C01761=-95.203,-21.462,17.374,-169.9520,-5.2148,-3137.2959
C01762=-94.842,-19.790,17.237,-164.8285,-6.4355,-3138.2136
C01763=-94.656,-17.748,17.095,-159.3411,-5.0626,-3139.3803
C01764=-94.777,-14.774,16.986,-155.9417,-1.9916,-3141.1399
C01765=-95.219,-10.339,16.941,-154.9335,-0.3011,-3143.8030
C01766=-95.617,-5.406,16.939,-154.8750,0.0274,-3146.7641
C01767=-95.772,0.000,16.941,-154.8879,-0.0000,-3150.0000
C01768=-95.617,5.406,16.939,-154.8750,-0.0274,-3153.2359
C01769=-95.219,10.339,16.941,-154.9335,0.3011,-3156.1970
C01770=-94.777,14.774,16.986,-155.9409,1.9854,-3158.8601
C01771=-94.656,17.748,17.095,-159.3411,5.0626,-3160.6197
C01772=-94.842,19.790,17.237,-164.8285,6.4355,-3161.7864
C01773=-95.203,21.462,17.374,-169.9520,5.2148,-3162.7041
C01774=-95.565,23.155,17.473,-173.2181,2.8849,-3163.6200
C01775=-95.708,25.257,17.521,-175.7539,1.0630,-3164.7831
C01776=-95.481,28.035,17.545,-178.1294,0.2806,-3166.3632
C01777=-94.884,31.135,17.565,-179.6411,0.0273,-3168.1666
C01778=-93.972,34.135,17.585,-179.9202,-0.0015,-3169.9634
C01779=-92.934,36.917,17.598,-179.9926,-0.0032,-3171.6649
C01780=-91.818,39.610,17.598,-179.9925,-0.0030,-3173.3352
C01781=-90.585,42.311,17.585,-179.9180,0.0004,-3175.0366
C01782=-89.109,45.077,17.565,-179.6386,-0.0291,-3176.8332
C01783=-87.339,47.692,17.545,-178.1307,-0.2787,-3178.6370
C01784=-85.535,49.816,17.521,-175.7503,-1.0646,-3180.2167
C01785=-83.948,51.202,17.473,-173.2162,-2.8847,-3181.3801
C01786=-82.495,52.143,17.374,-169.9475,-5.2185,-3182.2959
C01787=-81.058,53.070,17.237,-164.8269,-6.4371,-3183.2134
C01788=-79.482,54.382,17.095,-159.3399,-5.0676,-3184.3801
C01789=-77.464,56.571,16.986,-155.9409,-1.9875,-3186.1402
C01790=-74.640,60.019,16.941,-154.9325,-0.3004,-3188.8032
C01791=-71.434,63.789,16.939,-154.8745,0.0271,-3191.7642
C01792=-67.721,67.721,16.941,-154.8876,0.0000,-3195.0000
C01793=-63.789,71.434,16.939,-154.8745,-0.0271,-3198.2358
C01794=-60.019,74.640,16.941,-154.9325,0.3004,-3201.1968
C01795=-56.571,77.464,16.986,-155.9409,1.9875,-3203.8598
C01796=-54.382,79.482,17.095,-159.3399,5.0676,-3205.6199
C01797=-53.070,81.058,17.237,-164.8269,6.4371,-3206.7866
C01798=-52.143,82.495,17.374,-169.9475,5.2185,-3207.7041
C01799=-51.202,83.948,17.473,-173.2162,2.8847,-3208.6199
C01800=-49.816,85.535,17.521,-175.7503,1.0646,-3209.7833
C01801=-47.692,87.339,17.545,-178.1307,0.2787,-3211.3630
C01802=-45.077,89.109,17.565,-179.6386,0.0291,-3213.1668
C01803=-42.311,90.585,17.585,-179.9180,-0.0004,-3214.9634
C01804=-39.610,91.818,17.598,-179.9925,0.0030,-3216.6648
C01805=-36.917,92.934,17.598,-179.9926,0.0032,-3218.3351
C01806=-34.135,93.972,17.585,-179.9202,0.0015,-3220.0366
C01807=-31.135,94.884,17.565,-179.6411,-0.0273,-3221.8334
C01808=-28.035,95.481,17.545,-178.1294,-0.2806,-3223.6368
C01809=-25.257,95.708,17.521,-175.7539,-1.0630,-3225.2169
C01810=-23.155,95.565,17.473,-173.2181,-2.8849,-3226.3800
C01811=-21.462,95.203,17.374,-169.9520,-5.2148,-3227.2959
C01812=-19.790,94.842,17.237,-164.8285,-6.4355,-3228.2136
C01813=-17.748,94.656,17.095,-159.3411,-5.0626,-3229.3803
C01814=-14.774,94.777,16.986,-155.9409,-1.9854,-3231.1399
C01815=-10.339,95.219,16.941,-154.9335,-0.3011,-3233.8030
C01816=-5.406,95.617,16.939,-154.8750,0.0274,-3236.7641
C01817=0.000,95.772,16.941,-154.8879,-0.0000,-3240.0000
C01818=0.000,94.804,18.916,-152.9225,-0.0000,-3240.0000
C01819=5.317,94.652,18.914,-152.9126,-0.0298,-3243.2152
C01820=10.190,94.262,18.917,-152.9815,0.4089,-3246.1699
C01821=14.592,93.857,18.976,-154.1276,2.6863,-3248.8371
C01822=17.528,93.824,19.120,-158.3516,6.7345,-3250.5819
C01823=19.540,94.146,19.309,-165.0906,8.0389,-3251.7253
C01824=21.192,94.676,19.493,-170.7538,6.1439,-3252.6169
C01825=22.867,95.222,19.627,-173.7811,3.3954,-3253.5035
C01826=24.945,95.538,19.692,-175.9706,1.2792,-3254.6333
C01827=27.741,95.446,19.726,-178.2555,0.3221,-3256.2063
C01828=30.903,94.927,19.753,-179.7244,0.0234,-3258.0324
C01829=33.988,94.020,19.780,-179.9222,0.0038,-3259.8748
C01830=36.867,92.953,19.798,-179.9926,-0.0032,-3261.6343
C01831=39.659,91.796,19.798,-179.9925,-0.0030,-3263.3660
C01832=42.449,90.515,19.780,-179.9232,-0.0019,-3265.1253
C01833=45.272,88.975,19.753,-179.7282,-0.0288,-3266.9678
C01834=47.874,87.106,19.726,-178.2537,-0.3220,-3268.7935
C01835=49.917,85.194,19.692,-175.9742,-1.2794,-3270.3670
C01836=51.163,83.502,19.627,-173.7835,-3.3967,-3271.4965
C01837=51.961,81.931,19.493,-170.7560,-6.1455,-3272.3830
C01838=52.755,80.388,19.309,-165.0938,-8.0387,-3273.2751
C01839=53.950,78.738,19.120,-158.3479,-6.7340,-3274.4183
C01840=56.048,76.685,18.976,-154.1288,-2.6854,-3276.1625
C01841=59.448,73.859,18.917,-152.9797,-0.4094,-3278.8301
C01842=63.169,70.689,18.914,-152.9124,0.0356,-3281.7846
C01843=67.036,67.036,18.916,-152.9207,0.0000,-3285.0000
C01844=70.689,63.169,18.914,-152.9124,-0.0356,-3288.2154
C01845=73.859,59.448,18.917,-152.9797,0.4094,-3291.1699
C01846=76.685,56.048,18.976,-154.1288,2.6854,-3293.8375
C01847=78.738,53.950,19.120,-158.3479,6.7340,-3295.5817
C01848=80.388,52.755,19.309,-165.0938,8.0387,-3296.7249
C01849=81.931,51.961,19.493,-170.7560,6.1455,-3297.6170
C01850=83.502,51.163,19.627,-173.7835,3.3967,-3298.5035
C01851=85.194,49.917,19.692,-175.9742,1.2794,-3299.6330
C01852=87.106,47.874,19.726,-178.2537,0.3220,-3301.2065
C01853=88.975,45.272,19.753,-179.7282,0.0288,-3303.0322
C01854=90.515,42.449,19.780,-179.9232,0.0019,-3304.8747
C01855=91.796,39.659,19.798,-179.9925,0.0030,-3306.6340
C01856=92.953,36.867,19.798,-179.9926,0.0032,-3308.3657
C01857=94.020,33.988,19.780,-179.9222,-0.0038,-3310.1252
C01858=94.927,30.903,19.753,-179.7244,-0.0234,-3311.9676
C01859=95.446,27.741,19.726,-178.2555,-0.3221,-3313.7937
C01860=95.538,24.945,19.692,-175.9706,-1.2792,-3315.3667
C01861=95.222,22.867,19.627,-173.7811,-3.3954,-3316.4965
C01862=94.676,21.192,19.493,-170.7538,-6.1439,-3317.3831
C01863=94.146,19.540,19.309,-165.0906,-8.0389,-3318.2747
C01864=93.824,17.528,19.120,-158.3516,-6.7345,-3319.4181
C01865=93.857,14.592,18.976,-154.1276,-2.6863,-3321.1629
C01866=94.262,10.190,18.917,-152.9815,-0.4089,-3323.8301
C01867=94.652,5.317,18.914,-152.9126,0.0298,-3326.7848
C01868=94.804,0.000,18.916,-152.9225,-0.0000,-3330.0000
C01869=94.652,-5.317,18.914,-152.9126,-0.0298,-3333.2152
C01870=94.262,-10.190,18.917,-152.9815,0.4089,-3336.1699
C01871=93.857,-14.592,18.976,-154.1276,2.6863,-3338.8371
C01872=93.824,-17.528,19.120,-158.3516,6.7345,-3340.5819
C01873=94.146,-19.540,19.309,-165.0906,8.0389,-3341.7253
C01874=94.676,-21.192,19.493,-170.7538,6.1439,-3342.6169
C01875=95.222,-22.867,19.627,-173.7811,3.3954,-3343.5035
C01876=95.538,-24.945,19.692,-175.9706,1.2792,-3344.6333
C01877=95.446,-27.741,19.726,-178.2555,0.3221,-3346.2063
C01878=94.927,-30.903,19.753,-179.7244,0.0234,-3348.0324
C01879=94.020,-33.988,19.780,-179.9222,0.0038,-3349.8748
C01880=92.953,-36.867,19.798,-179.9926,-0.0032,-3351.6343
C01881=91.796,-39.659,19.798,-179.9925,-0.0030,-3353.3660
C01882=90.515,-42.449,19.780,-179.9232,-0.0019,-3355.1253
C01883=88.975,-45.272,19.753,-179.7282,-0.0288,-3356.9678
C01884=87.106,-47.874,19.726,-178.2537,-0.3220,-3358.7935
C01885=85.194,-49.917,19.692,-175.9742,-1.2794,-3360.3670
C01886=83.502,-51.163,19.627,-173.7835,-3.3967,-3361.4965
C01887=81.931,-51.961,19.493,-170.7560,-6.1455,-3362.3830
C01888=80.388,-52.755,19.309,-165.0938,-8.0387,-3363.2751
C01889=78.738,-53.950,19.120,-158.3479,-6.7340,-3364.4183
C01890=76.685,-56.048,18.976,-154.1288,-2.6854,-3366.1625
C01891=73.859,-59.448,18.917,-152.9797,-0.4094,-3368.8301
C01892=70.689,-63.169,18.914,-152.9124,0.0356,-3371.7846
C01893=67.036,-67.036,18.916,-152.9207,-0.0000,-3375.0000
C01894=63.169,-70.689,18.914,-152.9124,-0.0356,-3378.2154
C01895=59.448,-73.859,18.917,-152.9797,0.4094,-3381.1699
C01896=56.048,-76.685,18.976,-154.1288,2.6854,-3383.8375
C01897=53.950,-78.738,19.120,-158.3479,6.7340,-3385.5817
C01898=52.755,-80.388,19.309,-165.0938,8.0387,-3386.7249
C01899=51.961,-81.931,19.493,-170.7560,6.1455,-3387.6170
C01900=51.163,-83.502,19.627,-173.7835,3.3967,-3388.5035
C01901=49.917,-85.194,19.692,-175.9742,1.2794,-3389.6330
C01902=47.874,-87.106,19.726,-178.2537,0.3220,-3391.2065
C01903=45.272,-88.975,19.753,-179.7282,0.0288,-3393.0322
C01904=42.449,-90.515,19.780,-179.9232,0.0019,-3394.8747
C01905=39.659,-91.796,19.798,-179.9925,0.0030,-3396.6340
C01906=36.867,-92.953,19.798,-179.9926,0.0032,-3398.3657
C01907=33.988,-94.020,19.780,-179.9222,-0.0038,-3400.1252
C01908=30.903,-94.927,19.753,-179.7244,-0.0234,-3401.9676
C01909=27.741,-95.446,19.726,-178.2555,-0.3221,-3403.7937
C01910=24.945,-95.538,19.692,-175.9706,-1.2792,-3405.3667
C01911=22.867,-95.222,19.627,-173.7811,-3.3954,-3406.4965
C01912=21.192,-94.676,19.493,-170.7538,-6.1439,-3407.3831
C01913=19.540,-94.146,19.309,-165.0906,-8.0389,-3408.2747
C01914=17.528,-93.824,19.120,-158.3516,-6.7345,-3409.4181
C01915=14.592,-93.857,18.976,-154.1276,-2.6863,-3411.1629
C01916=10.190,-94.262,18.917,-152.9815,-0.4089,-3413.8301
C01917=5.317,-94.652,18.914,-152.9126,0.0298,-3416.7848
C01918=0.000,-94.804,18.916,-152.9225,0.0000,-3420.0000
C01919=0.000,-94.804,18.916,-152.9225,0.0000,-3420.0000
C01920=-5.317,-94.652,18.914,-152.9126,-0.0298,-3423.2152
C01921=-10.190,-94.262,18.917,-152.9815,0.4089,-3426.1699
C01922=-14.592,-93.857,18.976,-154.1276,2.6863,-3428.8371
C01923=-17.528,-93.824,19.120,-158.3516,6.7345,-3430.5819
C01924=-19.540,-94.146,19.309,-165.0906,8.0389,-3431.7253
C01925=-21.192,-94.676,19.493,-170.7538,6.1439,-3432.6169
C01926=-22.867,-95.222,19.627,-173.7811,3.3954,-3433.5035
C01927=-24.945,-95.538,19.692,-175.9706,1.2792,-3434.6333
C01928=-27.741,-95.446,19.726,-178.2555,0.3221,-3436.2063
C01929=-30.903,-94.927,19.753,-179.7244,0.0234,-3438.0324
C01930=-33.988,-94.020,19.780,-179.9222,0.0038,-3439.8748
C01931=-36.867,-92.953,19.798,-179.9926,-0.0032,-3441.6343
C01932=-39.659,-91.796,19.798,-179.9925,-0.0030,-3443.3660
C01933=-42.449,-90.515,19.780,-179.9232,-0.0019,-3445.1253
C01934=-45.272,-88.975,19.753,-179.7282,-0.0288,-3446.9678
C01935=-47.874,-87.106,19.726,-178.2537,-0.3220,-3448.7935
C01936=-49.917,-85.194,19.692,-175.9742,-1.2794,-3450.3670
C01937=-51.163,-83.502,19.627,-173.7835,-3.3967,-3451.4965
C01938=-51.961,-81.931,19.493,-170.7560,-6.1455,-3452.3830
C01939=-52.755,-80.388,19.309,-165.0938,-8.0387,-3453.2751
C01940=-53.950,-78.738,19.120,-158.3479,-6.7340,-3454.4183
C01941=-56.048,-76.685,18.976,-154.1288,-2.6854,-3456.1625
C01942=-59.448,-73.859,18.917,-152.9797,-0.4094,-3458.8301
C01943=-63.169,-70.689,18.914,-152.9124,0.0356,-3461.7846
C01944=-67.036,-67.036,18.916,-152.9207,-0.0000,-3465.0000
C01945=-70.689,-63.169,18.914,-152.9124,-0.0356,-3468.2154
C01946=-73.859,-59.448,18.917,-152.9797,0.4094,-3471.1699
C01947=-76.685,-56.048,18.976,-154.1288,2.6854,-3473.8375
C01948=-78.738,-53.950,19.120,-158.3479,6.7340,-3475.5817
C01949=-80.388,-52.755,19.309,-165.0938,8.0387,-3476.7249
C01950=-81.931,-51.961,19.493,-170.7560,6.1455,-3477.6170
C01951=-83.502,-51.163,19.627,-173.7835,3.3967,-3478.5035
C01952=-85.194,-49.917,19.692,-175.9742,1.2794,-3479.6330
C01953=-87.106,-47.874,19.726,-178.2537,0.3220,-3481.2065
C01954=-88.975,-45.272,19.753,-179.7282,0.0288,-3483.0322
C01955=-90.515,-42.449,19.780,-179.9232,0.0019,-3484.8747
C01956=-91.796,-39.659,19.798,-179.9925,0.0030,-3486.6340
C01957=-92.953,-36.867,19.798,-179.9926,0.0032,-3488.3657
C01958=-94.020,-33.988,19.780,-179.9222,-0.0038,-3490.1252
C01959=-94.927,-30.903,19.753,-179.7244,-0.0234,-3491.9676
C01960=-95.446,-27.741,19.726,-178.2555,-0.3221,-3493.7937
C01961=-95.538,-24.945,19.692,-175.9706,-1.2792,-3495.3667
C01962=-95.222,-22.867,19.627,-173.7811,-3.3954,-3496.4965
C01963=-94.676,-21.192,19.493,-170.7538,-6.1439,-3497.3831
C01964=-94.146,-19.540,19.309,-165.0906,-8.0389,-3498.2747
C01965=-93.824,-17.528,19.120,-158.3516,-6.7345,-3499.4181
C01966=-93.857,-14.592,18.976,-154.1276,-2.6863,-3501.1629
C01967=-94.262,-10.190,18.917,-152.9815,-0.4089,-3503.8301
C01968=-94.652,-5.317,18.914,-152.9126,0.0298,-3506.7848
C01969=-94.804,0.000,18.916,-152.9225,-0.0000,-3510.0000
C01970=-94.652,5.317,18.914,-152.9126,-0.0298,-3513.2152
C01971=-94.262,10.190,18.917,-152.9815,0.4089,-3516.1699
C01972=-93.857,14.592,18.976,-154.1276,2.6863,-3518.8371
C01973=-93.824,17.528,19.120,-158.3516,6.7345,-3520.5819
C01974=-94.146,19.540,19.309,-165.0906,8.0389,-3521.7253
C01975=-94.676,21.192,19.493,-170.7538,6.1439,-3522.6169
C01976=-95.222,22.867,19.627,-173.7811,3.3954,-3523.5035
C01977=-95.538,24.945,19.692,-175.9706,1.2792,-3524.6333
C01978=-95.446,27.741,19.726,-178.2555,0.3221,-3526.2063
C01979=-94.927,30.903,19.753,-179.7244,0.0234,-3528.0324
C01980=-94.020,33.988,19.780,-179.9222,0.0038,-3529.8748
C01981=-92.953,36.867,19.798,-179.9926,-0.0032,-3531.6343
C01982=-91.796,39.659,19.798,-179.9925,-0.0030,-3533.3660
C01983=-90.515,42.449,19.780,-179.9232,-0.0019,-3535.1253
C01984=-88.975,45.272,19.753,-179.7282,-0.0288,-3536.9678
C01985=-87.106,47.874,19.726,-178.2537,-0.3220,-3538.7935
C01986=-85.194,49.917,19.692,-175.9742,-1.2794,-3540.3670
C01987=-83.502,51.163,19.627,-173.7835,-3.3967,-3541.4965
C01988=-81.931,51.961,19.493,-170.7560,-6.1455,-3542.3830
C01989=-80.388,52.755,19.309,-165.0938,-8.0387,-3543.2751
C01990=-78.738,53.950,19.120,-158.3479,-6.7340,-3544.4183
C01991=-76.685,56.048,18.976,-154.1288,-2.6854,-3546.1625
C01992=-73.859,59.448,18.917,-152.9797,-0.4094,-3548.8301
C01993=-70.689,63.169,18.914,-152.9124,0.0356,-3551.7846
C01994=-67.036,67.036,18.916,-152.9207,0.0000,-3555.0000
C01995=-63.169,70.689,18.914,-152.9124,-0.0356,-3558.2154
C01996=-59.448,73.859,18.917,-152.9797,0.4094,-3561.1699
C01997=-56.048,76.685,18.976,-154.1288,2.6854,-3563.8375
C01998=-53.950,78.738,19.120,-158.3479,6.7340,-3565.5817
C01999=-52.755,80.388,19.309,-165.0938,8.0387,-3566.7249
///TOOL 0
///POSTYPE ANGLE
///ANGLE
EC00000=0.0000,0.0000
EC00001=0.0000,3.3204
EC00002=0.0000,6.3084
EC00003=0.0000,8.9540
EC00004=0.0000,10.7765
EC00005=0.0000,12.0369
EC00006=0.0000,13.0576
EC00007=0.0000,14.0938
EC00008=0.0000,15.3967
EC00009=0.0000,17.0065
EC00010=0.0000,18.7198
EC00011=0.0000,20.3278
EC00012=0.0000,21.7902
EC00013=0.0000,23.2098
EC00014=0.0000,24.6724
EC00015=0.0000,26.2801
EC00016=0.0000,27.9935
EC00017=0.0000,29.6039
EC00018=0.0000,30.9060
EC00019=0.0000,31.9421
EC00020=0.0000,32.9632
EC00021=0.0000,34.2234
EC00022=0.0000,36.0464
EC00023=0.0000,38.6909
EC00024=0.0000,41.6796
EC00025=0.0000,45.0000
EC00026=0.0000,48.3204
EC00027=0.0000,51.3091
EC00028=0.0000,53.9536
EC00029=0.0000,55.7766
EC00030=0.0000,57.0368
EC00031=0.0000,58.0579
EC00032=0.0000,59.0940
EC00033=0.0000,60.3961
EC00034=0.0000,62.0065
EC00035=0.0000,63.7199
EC00036=0.0000,65.3276
EC00037=0.0000,66.7902
EC00038=0.0000,68.2098
EC00039=0.0000,69.6722
EC00040=0.0000,71.2802
EC00041=0.0000,72.9935
EC00042=0.0000,74.6033
EC00043=0.0000,75.9062
EC00044=0.0000,76.9424
EC00045=0.0000,77.9631
EC00046=0.0000,79.2235
EC00047=0.0000,81.0460
EC00048=0.0000,83.6916
EC00049=0.0000,86.6796
EC00050=0.0000,90.0000
EC00051=0.0000,93.3204
EC00052=0.0000,96.3084
EC00053=0.0000,98.9540
EC00054=0.0000,100.7765
EC00055=0.0000,102.0369
EC00056=0.0000,103.0576
EC00057=0.0000,104.0938
EC00058=0.0000,105.3967
EC00059=0.0000,107.0065
EC00060=0.0000,108.7198
EC00061=0.0000,110.3278
EC00062=0.0000,111.7902
EC00063=0.0000,113.2098
EC00064=0.0000,114.6724
EC00065=0.0000,116.2801
EC00066=0.0000,117.9935
EC00067=0.0000,119.6039
EC00068=0.0000,120.9060
EC00069=0.0000,121.9421
EC00070=0.0000,122.9632
EC00071=0.0000,124.2234
EC00072=0.0000,126.0464
EC00073=0.0000,128.6909
EC00074=0.0000,131.6796
EC00075=0.0000,135.0000
EC00076=0.0000,138.3204
EC00077=0.0000,141.3091
EC00078=0.0000,143.9536
EC00079=0.0000,145.7766
EC00080=0.0000,147.0368
EC00081=0.0000,148.0579
EC00082=0.0000,149.0940
EC00083=0.0000,150.3961
EC00084=0.0000,152.0065
EC00085=0.0000,153.7199
EC00086=0.0000,155.3276
EC00087=0.0000,156.7902
EC00088=0.0000,158.2098
EC00089=0.0000,159.6722
EC00090=0.0000,161.2802
EC00091=0.0000,162.9935
EC00092=0.0000,164.6033
EC00093=0.0000,165.9062
EC00094=0.0000,166.9424
EC00095=0.0000,167.9631
EC00096=0.0000,169.2235
EC00097=0.0000,171.0460
EC00098=0.0000,173.6916
EC00099=0.0000,176.6796
EC00100=0.0000,180.0000
EC00101=0.0000,180.0000
EC00102=0.0000,183.3204
EC00103=0.0000,186.3084
EC00104=0.0000,188.9540
EC00105=0.0000,190.7765
EC00106=0.0000,192.0369
EC00107=0.0000,193.0576
EC00108=0.0000,194.0938
EC00109=0.0000,195.3967
EC00110=0.0000,197.0065
EC00111=0.0000,198.7198
EC00112=0.0000,200.3278
EC00113=0.0000,201.7902
EC00114=0.0000,203.2098
EC00115=0.0000,204.6724
EC00116=0.0000,206.2801
EC00117=0.0000,207.9935
EC00118=0.0000,209.6039
EC00119=0.0000,210.9060
EC00120=0.0000,211.9421
EC00121=0.0000,212.9632
EC00122=0.0000,214.2234
EC00123=0.0000,216.0464
EC00124=0.0000,218.6909
EC00125=0.0000,221.6796
EC00126=0.0000,225.0000
EC00127=0.0000,228.3204
EC00128=0.0000,231.3091
EC00129=0.0000,233.9536
EC00130=0.0000,235.7766
EC00131=0.0000,237.0368
EC00132=0.0000,238.0579
EC00133=0.0000,239.0940
EC00134=0.0000,240.3961
EC00135=0.0000,242.0065
EC00136=0.0000,243.7199
EC00137=0.0000,245.3276
EC00138=0.0000,246.7902
EC00139=0.0000,248.2098
EC00140=0.0000,249.6722
EC00141=0.0000,251.2802
EC00142=0.0000,252.9935
EC00143=0.0000,254.6033
EC00144=0.0000,255.9062
EC00145=0.0000,256.9424
EC00146=0.0000,257.9631
EC00147=0.0000,259.2235
EC00148=0.0000,261.0460
EC00149=0.0000,263.6916
EC00150=0.0000,266.6796
EC00151=0.0000,270.0000
EC00152=0.0000,273.3204
EC00153=0.0000,276.3084
EC00154=0.0000,278.9540
EC00155=0.0000,280.7765
EC00156=0.0000,282.0369
EC00157=0.0000,283.0576
EC00158=0.0000,284.0938
EC00159=0.0000,285.3967
EC00160=0.0000,287.0065
EC00161=0.0000,288.7198
EC00162=0.0000,290.3278
EC00163=0.0000,291.7902
EC00164=0.0000,293.2098
EC00165=0.0000,294.6724
EC00166=0.0000,296.2801
EC00167=0.0000,297.9935
EC00168=0.0000,299.6039
EC00169=0.0000,300.9060
EC00170=0.0000,301.9421
EC00171=0.0000,302.9632
EC00172=0.0000,304.2234
EC00173=0.0000,306.0464
EC00174=0.0000,308.6909
EC00175=0.0000,311.6796
EC00176=0.0000,315.0000
EC00177=0.0000,318.3204
EC00178=0.0000,321.3091
EC00179=0.0000,323.9536
EC00180=0.0000,325.7766
EC00181=0.0000,327.0368
EC00182=0.0000,328.0579
EC00183=0.0000,329.0940
EC00184=0.0000,330.3961
EC00185=0.0000,332.0065
EC00186=0.0000,333.7199
EC00187=0.0000,335.3276
EC00188=0.0000,336.7902
EC00189=0.0000,338.2098
EC00190=0.0000,339.6722
EC00191=0.0000,341.2802
EC00192=0.0000,342.9935
EC00193=0.0000,344.6033
EC00194=0.0000,345.9062
EC00195=0.0000,346.9424
EC00196=0.0000,347.9631
EC00197=0.0000,349.2235
EC00198=0.0000,351.0460
EC00199=0.0000,353.6916
EC00200=0.0000,356.6796
EC00201=0.0000,360.0000
EC00202=0.0000,360.0000
EC00203=0.0000,363.3190
EC00204=0.0000,366.3064
EC00205=0.0000,368.9521
EC00206=0.0000,370.7740
EC00207=0.0000,372.0325
EC00208=0.0000,373.0515
EC00209=0.0000,374.0856
EC00210=0.0000,375.3858
EC00211=0.0000,376.9948
EC00212=0.0000,378.7100
EC00213=0.0000,380.3211
EC00214=0.0000,381.7884
EC00215=0.0000,383.2118
EC00216=0.0000,384.6788
EC00217=0.0000,386.2904
EC00218=0.0000,388.0051
EC00219=0.0000,389.6142
EC00220=0.0000,390.9142
EC00221=0.0000,391.9485
EC00222=0.0000,392.9671
EC00223=0.0000,394.2260
EC00224=0.0000,396.0482
EC00225=0.0000,398.6933
EC00226=0.0000,401.6811
EC00227=0.0000,405.0000
EC00228=0.0000,408.3189
EC00229=0.0000,411.3067
EC00230=0.0000,413.9518
EC00231=0.0000,415.7740
EC00232=0.0000,417.0329
EC00233=0.0000,418.0515
EC00234=0.0000,419.0858
EC00235=0.0000,420.3858
EC00236=0.0000,421.9949
EC00237=0.0000,423.7096
EC00238=0.0000,425.3212
EC00239=0.0000,426.7882
EC00240=0.0000,428.2116
EC00241=0.0000,429.6789
EC00242=0.0000,431.2900
EC00243=0.0000,433.0052
EC00244=0.0000,434.6142
EC00245=0.0000,435.9144
EC00246=0.0000,436.9485
EC00247=0.0000,437.9675
EC00248=0.0000,439.2260
EC00249=0.0000,441.0479
EC00250=0.0000,443.6936
EC00251=0.0000,446.6810
EC00252=0.0000,450.0000
EC00253=0.0000,453.3190
EC00254=0.0000,456.3064
EC00255=0.0000,458.9521
EC00256=0.0000,460.7740
EC00257=0.0000,462.0325
EC00258=0.0000,463.0515
EC00259=0.0000,464.0856
EC00260=0.0000,465.3858
EC00261=0.0000,466.9948
EC00262=0.0000,468.7100
EC00263=0.0000,470.3211
EC00264=0.0000,471.7884
EC00265=0.0000,473.2118
EC00266=0.0000,474.6788
EC00267=0.0000,476.2904
EC00268=0.0000,478.0051
EC00269=0.0000,479.6142
EC00270=0.0000,480.9142
EC00271=0.0000,481.9485
EC00272=0.0000,482.9671
EC00273=0.0000,484.2260
EC00274=0.0000,486.0482
EC00275=0.0000,488.6933
EC00276=0.0000,491.6811
EC00277=0.0000,495.0000
EC00278=0.0000,498.3189
EC00279=0.0000,501.3067
EC00280=0.0000,503.9518
EC00281=0.0000,505.7740
EC00282=0.0000,507.0329
EC00283=0.0000,508.0515
EC00284=0.0000,509.0858
EC00285=0.0000,510.3858
EC00286=0.0000,511.9949
EC00287=0.0000,513.7096
EC00288=0.0000,515.3212
EC00289=0.0000,516.7882
EC00290=0.0000,518.2116
EC00291=0.0000,519.6789
EC00292=0.0000,521.2900
EC00293=0.0000,523.0052
EC00294=0.0000,524.6142
EC00295=0.0000,525.9144
EC00296=0.0000,526.9485
EC00297=0.0000,527.9675
EC00298=0.0000,529.2260
EC00299=0.0000,531.0479
EC00300=0.0000,533.6936
EC00301=0.0000,536.6810
EC00302=0.0000,540.0000
EC00303=0.0000,540.0000
EC00304=0.0000,543.3190
EC00305=0.0000,546.3064
EC00306=0.0000,548.9521
EC00307=0.0000,550.7740
EC00308=0.0000,552.0325
EC00309=0.0000,553.0515
EC00310=0.0000,554.0856
EC00311=0.0000,555.3858
EC00312=0.0000,556.9948
EC00313=0.0000,558.7100
EC00314=0.0000,560.3211
EC00315=0.0000,561.7884
EC00316=0.0000,563.2118
EC00317=0.0000,564.6788
EC00318=0.0000,566.2904
EC00319=0.0000,568.0051
EC00320=0.0000,569.6142
EC00321=0.0000,570.9142
EC00322=0.0000,571.9485
EC00323=0.0000,572.9671
EC00324=0.0000,574.2260
EC00325=0.0000,576.0482
EC00326=0.0000,578.6933
EC00327=0.0000,581.6811
EC00328=0.0000,585.0000
EC00329=0.0000,588.3189
EC00330=0.0000,591.3067
EC00331=0.0000,593.9518
EC00332=0.0000,595.7740
EC00333=0.0000,597.0329
EC00334=0.0000,598.0515
EC00335=0.0000,599.0858
EC00336=0.0000,600.3858
EC00337=0.0000,601.9949
EC00338=0.0000,603.7096
EC00339=0.0000,605.3212
EC00340=0.0000,606.7882
EC00341=0.0000,608.2116
EC00342=0.0000,609.6789
EC00343=0.0000,611.2900
EC00344=0.0000,613.0052
EC00345=0.0000,614.6142
EC00346=0.0000,615.9144
EC00347=0.0000,616.9485
EC00348=0.0000,617.9675
EC00349=0.0000,619.2260
EC00350=0.0000,621.0479
EC00351=0.0000,623.6936
EC00352=0.0000,626.6810
EC00353=0.0000,630.0000
EC00354=0.0000,633.3190
EC00355=0.0000,636.3064
EC00356=0.0000,638.9521
EC00357=0.0000,640.7740
EC00358=0.0000,642.0325
EC00359=0.0000,643.0515
EC00360=0.0000,644.0856
EC00361=0.0000,645.3858
EC00362=0.0000,646.9948
EC00363=0.0000,648.7100
EC00364=0.0000,650.3211
EC00365=0.0000,651.7884
EC00366=0.0000,653.2118
EC00367=0.0000,654.6788
EC00368=0.0000,656.2904
EC00369=0.0000,658.0051
EC00370=0.0000,659.6142
EC00371=0.0000,660.9142
EC00372=0.0000,661.9485
EC00373=0.0000,662.9671
EC00374=0.0000,664.2260
EC00375=0.0000,666.0482
EC00376=0.0000,668.6933
EC00377=0.0000,671.6811
EC00378=0.0000,675.0000
EC00379=0.0000,678.3189
EC00380=0.0000,681.3067
EC00381=0.0000,683.9518
EC00382=0.0000,685.7740
EC00383=0.0000,687.0329
EC00384=0.0000,688.0515
EC00385=0.0000,689.0858
EC00386=0.0000,690.3858
EC00387=0.0000,691.9949
EC00388=0.0000,693.7096
EC00389=0.0000,695.3212
EC00390=0.0000,696.7882
EC00391=0.0000,698.2116
EC00392=0.0000,699.6789
EC00393=0.0000,701.2900
EC00394=0.0000,703.0052
EC00395=0.0000,704.6142
EC00396=0.0000,705.9144
EC00397=0.0000,706.9485
EC00398=0.0000,707.9675
EC00399=0.0000,709.2260
EC00400=0.0000,711.0479
EC00401=0.0000,713.6936
EC00402=0.0000,716.6810
EC00403=0.0000,720.0000
EC00404=0.0000,720.0000
EC00405=0.0000,723.3146
EC00406=0.0000,726.3008
EC00407=0.0000,728.9471
EC00408=0.0000,730.7659
EC00409=0.0000,732.0199
EC00410=0.0000,733.0335
EC00411=0.0000,734.0616
EC00412=0.0000,735.3544
EC00413=0.0000,736.9622
EC00414=0.0000,738.6812
EC00415=0.0000,740.3024
EC00416=0.0000,741.7817
EC00417=0.0000,743.2185
EC00418=0.0000,744.6975
EC00419=0.0000,746.3188
EC00420=0.0000,748.0383
EC00421=0.0000,749.6456
EC00422=0.0000,750.9386
EC00423=0.0000,751.9667
EC00424=0.0000,752.9801
EC00425=0.0000,754.2340
EC00426=0.0000,756.0529
EC00427=0.0000,758.6992
EC00428=0.0000,761.6856
EC00429=0.0000,765.0000
EC00430=0.0000,768.3144
EC00431=0.0000,771.3008
EC00432=0.0000,773.9471
EC00433=0.0000,775.7660
EC00434=0.0000,777.0199
EC00435=0.0000,778.0333
EC00436=0.0000,779.0614
EC00437=0.0000,780.3544
EC00438=0.0000,781.9617
EC00439=0.0000,783.6812
EC00440=0.0000,785.3025
EC00441=0.0000,786.7815
EC00442=0.0000,788.2183
EC00443=0.0000,789.6976
EC00444=0.0000,791.3188
EC00445=0.0000,793.0378
EC00446=0.0000,794.6456
EC00447=0.0000,795.9384
EC00448=0.0000,796.9665
EC00449=0.0000,797.9801
EC00450=0.0000,799.2341
EC00451=0.0000,801.0529
EC00452=0.0000,803.6992
EC00453=0.0000,806.6854
EC00454=0.0000,810.0000
EC00455=0.0000,813.3146
EC00456=0.0000,816.3008
EC00457=0.0000,818.9471
EC00458=0.0000,820.7659
EC00459=0.0000,822.0199
EC00460=0.0000,823.0335
EC00461=0.0000,824.0616
EC00462=0.0000,825.3544
EC00463=0.0000,826.9622
EC00464=0.0000,828.6812
EC00465=0.0000,830.3024
EC00466=0.0000,831.7817
EC00467=0.0000,833.2185
EC00468=0.0000,834.6975
EC00469=0.0000,836.3188
EC00470=0.0000,838.0383
EC00471=0.0000,839.6456
EC00472=0.0000,840.9386
EC00473=0.0000,841.9667
EC00474=0.0000,842.9801
EC00475=0.0000,844.2340
EC00476=0.0000,846.0529
EC00477=0.0000,848.6992
EC00478=0.0000,851.6856
EC00479=0.0000,855.0000
EC00480=0.0000,858.3144
EC00481=0.0000,861.3008
EC00482=0.0000,863.9471
EC00483=0.0000,865.7660
EC00484=0.0000,867.0199
EC00485=0.0000,868.0333
EC00486=0.0000,869.0614
EC00487=0.0000,870.3544
EC00488=0.0000,871.9617
EC00489=0.0000,873.6812
EC00490=0.0000,875.3025
EC00491=0.0000,876.7815
EC00492=0.0000,878.2183
EC00493=0.0000,879.6976
EC00494=0.0000,881.3188
EC00495=0.0000,883.0378
EC00496=0.0000,884.6456
EC00497=0.0000,885.9384
EC00498=0.0000,886.9665
EC00499=0.0000,887.9801
EC00500=0.0000,889.2341
EC00501=0.0000,891.0529
EC00502=0.0000,893.6992
EC00503=0.0000,896.6854
EC00504=0.0000,900.0000
EC00505=0.0000,900.0000
EC00506=0.0000,903.3146
EC00507=0.0000,906.3008
EC00508=0.0000,908.9471
EC00509=0.0000,910.7659
EC00510=0.0000,912.0199
EC00511=0.0000,913.0335
EC00512=0.0000,914.0616
EC00513=0.0000,915.3544
EC00514=0.0000,916.9622
EC00515=0.0000,918.6812
EC00516=0.0000,920.3024
EC00517=0.0000,921.7817
EC00518=0.0000,923.2185
EC00519=0.0000,924.6975
EC00520=0.0000,926.3188
EC00521=0.0000,928.0383
EC00522=0.0000,929.6456
EC00523=0.0000,930.9386
EC00524=0.0000,931.9667
EC00525=0.0000,932.9801
EC00526=0.0000,934.2340
EC00527=0.0000,936.0529
EC00528=0.0000,938.6992
EC00529=0.0000,941.6856
EC00530=0.0000,945.0000
EC00531=0.0000,948.3144
EC00532=0.0000,951.3008
EC00533=0.0000,953.9471
EC00534=0.0000,955.7660
EC00535=0.0000,957.0199
EC00536=0.0000,958.0333
EC00537=0.0000,959.0614
EC00538=0.0000,960.3544
EC00539=0.0000,961.9617
EC00540=0.0000,963.6812
EC00541=0.0000,965.3025
EC00542=0.0000,966.7815
EC00543=0.0000,968.2183
EC00544=0.0000,969.6976
EC00545=0.0000,971.3188
EC00546=0.0000,973.0378
EC00547=0.0000,974.6456
EC00548=0.0000,975.9384
EC00549=0.0000,976.9665
EC00550=0.0000,977.9801
EC00551=0.0000,979.2341
EC00552=0.0000,981.0529
EC00553=0.0000,983.6992
EC00554=0.0000,986.6854
EC00555=0.0000,990.0000
EC00556=0.0000,993.3146
EC00557=0.0000,996.3008
EC00558=0.0000,998.9471
EC00559=0.0000,1000.7659
EC00560=0.0000,1002.0199
EC00561=0.0000,1003.0335
EC00562=0.0000,1004.0616
EC00563=0.0000,1005.3544
EC00564=0.0000,1006.9622
EC00565=0.0000,1008.6812
EC00566=0.0000,1010.3024
EC00567=0.0000,1011.7817
EC00568=0.0000,1013.2185
EC00569=0.0000,1014.6975
EC00570=0.0000,1016.3188
EC00571=0.0000,1018.0383
EC00572=0.0000,1019.6456
EC00573=0.0000,1020.9386
EC00574=0.0000,1021.9667
EC00575=0.0000,1022.9801
EC00576=0.0000,1024.2340
EC00577=0.0000,1026.0529
EC00578=0.0000,1028.6992
EC00579=0.0000,1031.6856
EC00580=0.0000,1035.0000
EC00581=0.0000,1038.3144
EC00582=0.0000,1041.3008
EC00583=0.0000,1043.9471
EC00584=0.0000,1045.7660
EC00585=0.0000,1047.0199
EC00586=0.0000,1048.0333
EC00587=0.0000,1049.0614
EC00588=0.0000,1050.3544
EC00589=0.0000,1051.9617
EC00590=0.0000,1053.6812
EC00591=0.0000,1055.3025
EC00592=0.0000,1056.7815
EC00593=0.0000,1058.2183
EC00594=0.0000,1059.6976
EC00595=0.0000,1061.3188
EC00596=0.0000,1063.0378
EC00597=0.0000,1064.6456
EC00598=0.0000,1065.9384
EC00599=0.0000,1066.9665
EC00600=0.0000,1067.9801
EC00601=0.0000,1069.2341
EC00602=0.0000,1071.0529
EC00603=0.0000,1073.6992
EC00604=0.0000,1076.6854
EC00605=0.0000,1080.0000
EC00606=0.0000,1080.0000
EC00607=0.0000,1083.3073
EC00608=0.0000,1086.2913
EC00609=0.0000,1088.9391
EC00610=0.0000,1090.7524
EC00611=0.0000,1091.9986
EC00612=0.0000,1093.0036
EC00613=0.0000,1094.0220
EC00614=0.0000,1095.3030
EC00615=0.0000,1096.9082
EC00616=0.0000,1098.6350
EC00617=0.0000,1100.2716
EC00618=0.0000,1101.7712
EC00619=0.0000,1103.2288
EC00620=0.0000,1104.7282
EC00621=0.0000,1106.3649
EC00622=0.0000,1108.0920
EC00623=0.0000,1109.6973
EC00624=0.0000,1110.9780
EC00625=0.0000,1111.9962
EC00626=0.0000,1113.0013
EC00627=0.0000,1114.2478
EC00628=0.0000,1116.0610
EC00629=0.0000,1118.7088
EC00630=0.0000,1121.6924
EC00631=0.0000,1125.0000
EC00632=0.0000,1128.3076
EC00633=0.0000,1131.2912
EC00634=0.0000,1133.9390
EC00635=0.0000,1135.7522
EC00636=0.0000,1136.9987
EC00637=0.0000,1138.0038
EC00638=0.0000,1139.0220
EC00639=0.0000,1140.3027
EC00640=0.0000,1141.9080
EC00641=0.0000,1143.6351
EC00642=0.0000,1145.2718
EC00643=0.0000,1146.7712
EC00644=0.0000,1148.2288
EC00645=0.0000,1149.7284
EC00646=0.0000,1151.3650
EC00647=0.0000,1153.0918
EC00648=0.0000,1154.6970
EC00649=0.0000,1155.9780
EC00650=0.0000,1156.9964
EC00651=0.0000,1158.0014
EC00652=0.0000,1159.2476
EC00653=0.0000,1161.0609
EC00654=0.0000,1163.7087
EC00655=0.0000,1166.6927
EC00656=0.0000,1170.0000
EC00657=0.0000,1173.3073
EC00658=0.0000,1176.2913
EC00659=0.0000,1178.9391
EC00660=0.0000,1180.7524
EC00661=0.0000,1181.9986
EC00662=0.0000,1183.0036
EC00663=0.0000,1184.0220
EC00664=0.0000,1185.3030
EC00665=0.0000,1186.9082
EC00666=0.0000,1188.6350
EC00667=0.0000,1190.2716
EC00668=0.0000,1191.7712
EC00669=0.0000,1193.2288
EC00670=0.0000,1194.7282
EC00671=0.0000,1196.3649
EC00672=0.0000,1198.0920
EC00673=0.0000,1199.6973
EC00674=0.0000,1200.9780
EC00675=0.0000,1201.9962
EC00676=0.0000,1203.0013
EC00677=0.0000,1204.2478
EC00678=0.0000,1206.0610
EC00679=0.0000,1208.7088
EC00680=0.0000,1211.6924
EC00681=0.0000,1215.0000
EC00682=0.0000,1218.3076
EC00683=0.0000,1221.2912
EC00684=0.0000,1223.9390
EC00685=0.0000,1225.7522
EC00686=0.0000,1226.9987
EC00687=0.0000,1228.0038
EC00688=0.0000,1229.0220
EC00689=0.0000,1230.3027
EC00690=0.0000,1231.9080
EC00691=0.0000,1233.6351
EC00692=0.0000,1235.2718
EC00693=0.0000,1236.7712
EC00694=0.0000,1238.2288
EC00695=0.0000,1239.7284
EC00696=0.0000,1241.3650
EC00697=0.0000,1243.0918
EC00698=0.0000,1244.6970
EC00699=0.0000,1245.9780
EC00700=0.0000,1246.9964
EC00701=0.0000,1248.0014
EC00702=0.0000,1249.2476
EC00703=0.0000,1251.0609
EC00704=0.0000,1253.7087
EC00705=0.0000,1256.6927
EC00706=0.0000,1260.0000
EC00707=0.0000,1260.0000
EC00708=0.0000,1263.3073
EC00709=0.0000,1266.2913
EC00710=0.0000,1268.9391
EC00711=0.0000,1270.7524
EC00712=0.0000,1271.9986
EC00713=0.0000,1273.0036
EC00714=0.0000,1274.0220
EC00715=0.0000,1275.3030
EC00716=0.0000,1276.9082
EC00717=0.0000,1278.6350
EC00718=0.0000,1280.2716
EC00719=0.0000,1281.7712
EC00720=0.0000,1283.2288
EC00721=0.0000,1284.7282
EC00722=0.0000,1286.3649
EC00723=0.0000,1288.0920
EC00724=0.0000,1289.6973
EC00725=0.0000,1290.9780
EC00726=0.0000,1291.9962
EC00727=0.0000,1293.0013
EC00728=0.0000,1294.2478
EC00729=0.0000,1296.0610
EC00730=0.0000,1298.7088
EC00731=0.0000,1301.6924
EC00732=0.0000,1305.0000
EC00733=0.0000,1308.3076
EC00734=0.0000,1311.2912
EC00735=0.0000,1313.9390
EC00736=0.0000,1315.7522
EC00737=0.0000,1316.9987
EC00738=0.0000,1318.0038
EC00739=0.0000,1319.0220
EC00740=0.0000,1320.3027
EC00741=0.0000,1321.9080
EC00742=0.0000,1323.6351
EC00743=0.0000,1325.2718
EC00744=0.0000,1326.7712
EC00745=0.0000,1328.2288
EC00746=0.0000,1329.7284
EC00747=0.0000,1331.3650
EC00748=0.0000,1333.0918
EC00749=0.0000,1334.6970
EC00750=0.0000,1335.9780
EC00751=0.0000,1336.9964
EC00752=0.0000,1338.0014
EC00753=0.0000,1339.2476
EC00754=0.0000,1341.0609
EC00755=0.0000,1343.7087
EC00756=0.0000,1346.6927
EC00757=0.0000,1350.0000
EC00758=0.0000,1353.3073
EC00759=0.0000,1356.2913
EC00760=0.0000,1358.9391
EC00761=0.0000,1360.7524
EC00762=0.0000,1361.9986
EC00763=0.0000,1363.0036
EC00764=0.0000,1364.0220
EC00765=0.0000,1365.3030
EC00766=0.0000,1366.9082
EC00767=0.0000,1368.6350
EC00768=0.0000,1370.2716
EC00769=0.0000,1371.7712
EC00770=0.0000,1373.2288
EC00771=0.0000,1374.7282
EC00772=0.0000,1376.3649
EC00773=0.0000,1378.0920
EC00774=0.0000,1379.6973
EC00775=0.0000,1380.9780
EC00776=0.0000,1381.9962
EC00777=0.0000,1383.0013
EC00778=0.0000,1384.2478
EC00779=0.0000,1386.0610
EC00780=0.0000,1388.7088
EC00781=0.0000,1391.6924
EC00782=0.0000,1395.0000
EC00783=0.0000,1398.3076
EC00784=0.0000,1401.2912
EC00785=0.0000,1403.9390
EC00786=0.0000,1405.7522
EC00787=0.0000,1406.9987
EC00788=0.0000,1408.0038
EC00789=0.0000,1409.0220
EC00790=0.0000,1410.3027
EC00791=0.0000,1411.9080
EC00792=0.0000,1413.6351
EC00793=0.0000,1415.2718
EC00794=0.0000,1416.7712
EC00795=0.0000,1418.2288
EC00796=0.0000,1419.7284
EC00797=0.0000,1421.3650
EC00798=0.0000,1423.0918
EC00799=0.0000,1424.6970
EC00800=0.0000,1425.9780
EC00801=0.0000,1426.9964
EC00802=0.0000,1428.0014
EC00803=0.0000,1429.2476
EC00804=0.0000,1431.0609
EC00805=0.0000,1433.7087
EC00806=0.0000,1436.6927
EC00807=0.0000,1440.0000
EC00808=0.0000,1440.0000
EC00809=0.0000,1443.2974
EC00810=0.0000,1446.2783
EC00811=0.0000,1448.9284
EC00812=0.0000,1450.7347
EC00813=0.0000,1451.9700
EC00814=0.0000,1452.9633
EC00815=0.0000,1453.9678
EC00816=0.0000,1455.2327
EC00817=0.0000,1456.8342
EC00818=0.0000,1458.5716
EC00819=0.0000,1460.2300
EC00820=0.0000,1461.7565
EC00821=0.0000,1463.2431
EC00822=0.0000,1464.7700
EC00823=0.0000,1466.4284
EC00824=0.0000,1468.1658
EC00825=0.0000,1469.7669
EC00826=0.0000,1471.0323
EC00827=0.0000,1472.0364
EC00828=0.0000,1473.0299
EC00829=0.0000,1474.2655
EC00830=0.0000,1476.0719
EC00831=0.0000,1478.7215
EC00832=0.0000,1481.7023
EC00833=0.0000,1485.0000
EC00834=0.0000,1488.2977
EC00835=0.0000,1491.2785
EC00836=0.0000,1493.9281
EC00837=0.0000,1495.7345
EC00838=0.0000,1496.9701
EC00839=0.0000,1497.9636
EC00840=0.0000,1498.9677
EC00841=0.0000,1500.2331
EC00842=0.0000,1501.8342
EC00843=0.0000,1503.5716
EC00844=0.0000,1505.2300
EC00845=0.0000,1506.7569
EC00846=0.0000,1508.2435
EC00847=0.0000,1509.7700
EC00848=0.0000,1511.4284
EC00849=0.0000,1513.1658
EC00850=0.0000,1514.7673
EC00851=0.0000,1516.0322
EC00852=0.0000,1517.0367
EC00853=0.0000,1518.0300
EC00854=0.0000,1519.2653
EC00855=0.0000,1521.0716
EC00856=0.0000,1523.7217
EC00857=0.0000,1526.7026
EC00858=0.0000,1530.0000
EC00859=0.0000,1533.2974
EC00860=0.0000,1536.2783
EC00861=0.0000,1538.9284
EC00862=0.0000,1540.7347
EC00863=0.0000,1541.9700
EC00864=0.0000,1542.9633
EC00865=0.0000,1543.9678
EC00866=0.0000,1545.2327
EC00867=0.0000,1546.8342
EC00868=0.0000,1548.5716
EC00869=0.0000,1550.2300
EC00870=0.0000,1551.7565
EC00871=0.0000,1553.2431
EC00872=0.0000,1554.7700
EC00873=0.0000,1556.4284
EC00874=0.0000,1558.1658
EC00875=0.0000,1559.7669
EC00876=0.0000,1561.0323
EC00877=0.0000,1562.0364
EC00878=0.0000,1563.0299
EC00879=0.0000,1564.2655
EC00880=0.0000,1566.0719
EC00881=0.0000,1568.7215
EC00882=0.0000,1571.7023
EC00883=0.0000,1575.0000
EC00884=0.0000,1578.2977
EC00885=0.0000,1581.2785
EC00886=0.0000,1583.9281
EC00887=0.0000,1585.7345
EC00888=0.0000,1586.9701
EC00889=0.0000,1587.9636
EC00890=0.0000,1588.9677
EC00891=0.0000,1590.2331
EC00892=0.0000,1591.8342
EC00893=0.0000,1593.5716
EC00894=0.0000,1595.2300
EC00895=0.0000,1596.7569
EC00896=0.0000,1598.2435
EC00897=0.0000,1599.7700
EC00898=0.0000,1601.4284
EC00899=0.0000,1603.1658
EC00900=0.0000,1604.7673
EC00901=0.0000,1606.0322
EC00902=0.0000,1607.0367
EC00903=0.0000,1608.0300
EC00904=0.0000,1609.2653
EC00905=0.0000,1611.0716
EC00906=0.0000,1613.7217
EC00907=0.0000,1616.7026
EC00908=0.0000,1620.0000
EC00909=0.0000,1620.0000
EC00910=0.0000,1623.2974
EC00911=0.0000,1626.2783
EC00912=0.0000,1628.9284
EC00913=0.0000,1630.7347
EC00914=0.0000,1631.9700
EC00915=0.0000,1632.9633
EC00916=0.0000,1633.9678
EC00917=0.0000,1635.2327
EC00918=0.0000,1636.8342
EC00919=0.0000,1638.5716
EC00920=0.0000,1640.2300
EC00921=0.0000,1641.7565
EC00922=0.0000,1643.2431
EC00923=0.0000,1644.7700
EC00924=0.0000,1646.4284
EC00925=0.0000,1648.1658
EC00926=0.0000,1649.7669
EC00927=0.0000,1651.0323
EC00928=0.0000,1652.0364
EC00929=0.0000,1653.0299
EC00930=0.0000,1654.2655
EC00931=0.0000,1656.0719
EC00932=0.0000,1658.7215
EC00933=0.0000,1661.7023
EC00934=0.0000,1665.0000
EC00935=0.0000,1668.2977
EC00936=0.0000,1671.2785
EC00937=0.0000,1673.9281
EC00938=0.0000,1675.7345
EC00939=0.0000,1676.9701
EC00940=0.0000,1677.9636
EC00941=0.0000,1678.9677
EC00942=0.0000,1680.2331
EC00943=0.0000,1681.8342
EC00944=0.0000,1683.5716
EC00945=0.0000,1685.2300
EC00946=0.0000,1686.7569
EC00947=0.0000,1688.2435
EC00948=0.0000,1689.7700
EC00949=0.0000,1691.4284
EC00950=0.0000,1693.1658
EC00951=0.0000,1694.7673
EC00952=0.0000,1696.0322
EC00953=0.0000,1697.0367
EC00954=0.0000,1698.0300
EC00955=0.0000,1699.2653
EC00956=0.0000,1701.0716
EC00957=0.0000,1703.7217
EC00958=0.0000,1706.7026
EC00959=0.0000,1710.0000
EC00960=0.0000,1713.2974
EC00961=0.0000,1716.2783
EC00962=0.0000,1718.9284
EC00963=0.0000,1720.7347
EC00964=0.0000,1721.9700
EC00965=0.0000,1722.9633
EC00966=0.0000,1723.9678
EC00967=0.0000,1725.2327
EC00968=0.0000,1726.8342
EC00969=0.0000,1728.5716
EC00970=0.0000,1730.2300
EC00971=0.0000,1731.7565
EC00972=0.0000,1733.2431
EC00973=0.0000,1734.7700
EC00974=0.0000,1736.4284
EC00975=0.0000,1738.1658
EC00976=0.0000,1739.7669
EC00977=0.0000,1741.0323
EC00978=0.0000,1742.0364
EC00979=0.0000,1743.0299
EC00980=0.0000,1744.2655
EC00981=0.0000,1746.0719
EC00982=0.0000,1748.7215
EC00983=0.0000,1751.7023
EC00984=0.0000,1755.0000
EC00985=0.0000,1758.2977
EC00986=0.0000,1761.2785
EC00987=0.0000,1763.9281
EC00988=0.0000,1765.7345
EC00989=0.0000,1766.9701
EC00990=0.0000,1767.9636
EC00991=0.0000,1768.9677
EC00992=0.0000,1770.2331
EC00993=0.0000,1771.8342
EC00994=0.0000,1773.5716
EC00995=0.0000,1775.2300
EC00996=0.0000,1776.7569
EC00997=0.0000,1778.2435
EC00998=0.0000,1779.7700
EC00999=0.0000,1781.4284
EC01000=0.0000,1783.1658
EC01001=0.0000,1784.7673
EC01002=0.0000,1786.0322
EC01003=0.0000,1787.0367
EC01004=0.0000,1788.0300
EC01005=0.0000,1789.2653
EC01006=0.0000,1791.0716
EC01007=0.0000,1793.7217
EC01008=0.0000,1796.7026
EC01009=0.0000,1800.0000
EC01010=0.0000,1800.0000
EC01011=0.0000,1803.2854
EC01012=0.0000,1806.2621
EC01013=0.0000,1808.9150
EC01014=0.0000,1810.7121
EC01015=0.0000,1811.9342
EC01016=0.0000,1812.9128
EC01017=0.0000,1813.8997
EC01018=0.0000,1815.1448
EC01019=0.0000,1816.7421
EC01020=0.0000,1818.4921
EC01021=0.0000,1820.1777
EC01022=0.0000,1821.7387
EC01023=0.0000,1823.2613
EC01024=0.0000,1824.8225
EC01025=0.0000,1826.5076
EC01026=0.0000,1828.2578
EC01027=0.0000,1829.8549
EC01028=0.0000,1831.1001
EC01029=0.0000,1832.0874
EC01030=0.0000,1833.0661
EC01031=0.0000,1834.2883
EC01032=0.0000,1836.0850
EC01033=0.0000,1838.7375
EC01034=0.0000,1841.7146
EC01035=0.0000,1845.0000
EC01036=0.0000,1848.2854
EC01037=0.0000,1851.2625
EC01038=0.0000,1853.9150
EC01039=0.0000,1855.7117
EC01040=0.0000,1856.9339
EC01041=0.0000,1857.9126
EC01042=0.0000,1858.8999
EC01043=0.0000,1860.1451
EC01044=0.0000,1861.7422
EC01045=0.0000,1863.4924
EC01046=0.0000,1865.1775
EC01047=0.0000,1866.7387
EC01048=0.0000,1868.2613
EC01049=0.0000,1869.8223
EC01050=0.0000,1871.5079
EC01051=0.0000,1873.2579
EC01052=0.0000,1874.8552
EC01053=0.0000,1876.1003
EC01054=0.0000,1877.0872
EC01055=0.0000,1878.0658
EC01056=0.0000,1879.2879
EC01057=0.0000,1881.0850
EC01058=0.0000,1883.7379
EC01059=0.0000,1886.7146
EC01060=0.0000,1890.0000
EC01061=0.0000,1893.2854
EC01062=0.0000,1896.2621
EC01063=0.0000,1898.9150
EC01064=0.0000,1900.7121
EC01065=0.0000,1901.9342
EC01066=0.0000,1902.9128
EC01067=0.0000,1903.8997
EC01068=0.0000,1905.1448
EC01069=0.0000,1906.7421
EC01070=0.0000,1908.4921
EC01071=0.0000,1910.1777
EC01072=0.0000,1911.7387
EC01073=0.0000,1913.2613
EC01074=0.0000,1914.8225
EC01075=0.0000,1916.5076
EC01076=0.0000,1918.2578
EC01077=0.0000,1919.8549
EC01078=0.0000,1921.1001
EC01079=0.0000,1922.0874
EC01080=0.0000,1923.0661
EC01081=0.0000,1924.2883
EC01082=0.0000,1926.0850
EC01083=0.0000,1928.7375
EC01084=0.0000,1931.7146
EC01085=0.0000,1935.0000
EC01086=0.0000,1938.2854
EC01087=0.0000,1941.2625
EC01088=0.0000,1943.9150
EC01089=0.0000,1945.7117
EC01090=0.0000,1946.9339
EC01091=0.0000,1947.9126
EC01092=0.0000,1948.8999
EC01093=0.0000,1950.1451
EC01094=0.0000,1951.7422
EC01095=0.0000,1953.4924
EC01096=0.0000,1955.1775
EC01097=0.0000,1956.7387
EC01098=0.0000,1958.2613
EC01099=0.0000,1959.8223
EC01100=0.0000,1961.5079
EC01101=0.0000,1963.2579
EC01102=0.0000,1964.8552
EC01103=0.0000,1966.1003
EC01104=0.0000,1967.0872
EC01105=0.0000,1968.0658
EC01106=0.0000,1969.2879
EC01107=0.0000,1971.0850
EC01108=0.0000,1973.7379
EC01109=0.0000,1976.7146
EC01110=0.0000,1980.0000
EC01111=0.0000,1980.0000
EC01112=0.0000,1983.2854
EC01113=0.0000,1986.2621
EC01114=0.0000,1988.9150
EC01115=0.0000,1990.7121
EC01116=0.0000,1991.9342
EC01117=0.0000,1992.9128
EC01118=0.0000,1993.8997
EC01119=0.0000,1995.1448
EC01120=0.0000,1996.7421
EC01121=0.0000,1998.4921
EC01122=0.0000,2000.1777
EC01123=0.0000,2001.7387
EC01124=0.0000,2003.2613
EC01125=0.0000,2004.8225
EC01126=0.0000,2006.5076
EC01127=0.0000,2008.2578
EC01128=0.0000,2009.8549
EC01129=0.0000,2011.1001
EC01130=0.0000,2012.0874
EC01131=0.0000,2013.0661
EC01132=0.0000,2014.2883
EC01133=0.0000,2016.0850
EC01134=0.0000,2018.7375
EC01135=0.0000,2021.7146
EC01136=0.0000,2025.0000
EC01137=0.0000,2028.2854
EC01138=0.0000,2031.2625
EC01139=0.0000,2033.9150
EC01140=0.0000,2035.7117
EC01141=0.0000,2036.9339
EC01142=0.0000,2037.9126
EC01143=0.0000,2038.8999
EC01144=0.0000,2040.1451
EC01145=0.0000,2041.7422
EC01146=0.0000,2043.4924
EC01147=0.0000,2045.1775
EC01148=0.0000,2046.7387
EC01149=0.0000,2048.2613
EC01150=0.0000,2049.8223
EC01151=0.0000,2051.5079
EC01152=0.0000,2053.2579
EC01153=0.0000,2054.8552
EC01154=0.0000,2056.1003
EC01155=0.0000,2057.0872
EC01156=0.0000,2058.0658
EC01157=0.0000,2059.2879
EC01158=0.0000,2061.0850
EC01159=0.0000,2063.7379
EC01160=0.0000,2066.7146
EC01161=0.0000,2070.0000
EC01162=0.0000,2073.2854
EC01163=0.0000,2076.2621
EC01164=0.0000,2078.9150
EC01165=0.0000,2080.7121
EC01166=0.0000,2081.9342
EC01167=0.0000,2082.9128
EC01168=0.0000,2083.8997
EC01169=0.0000,2085.1448
EC01170=0.0000,2086.7421
EC01171=0.0000,2088.4921
EC01172=0.0000,2090.1777
EC01173=0.0000,2091.7387
EC01174=0.0000,2093.2613
EC01175=0.0000,2094.8225
EC01176=0.0000,2096.5076
EC01177=0.0000,2098.2578
EC01178=0.0000,2099.8549
EC01179=0.0000,2101.1001
EC01180=0.0000,2102.0874
EC01181=0.0000,2103.0661
EC01182=0.0000,2104.2883
EC01183=0.0000,2106.0850
EC01184=0.0000,2108.7375
EC01185=0.0000,2111.7146
EC01186=0.0000,2115.0000
EC01187=0.0000,2118.2854
EC01188=0.0000,2121.2625
EC01189=0.0000,2123.9150
EC01190=0.0000,2125.7117
EC01191=0.0000,2126.9339
EC01192=0.0000,2127.9126
EC01193=0.0000,2128.8999
EC01194=0.0000,2130.1451
EC01195=0.0000,2131.7422
EC01196=0.0000,2133.4924
EC01197=0.0000,2135.1775
EC01198=0.0000,2136.7387
EC01199=0.0000,2138.2613
EC01200=0.0000,2139.8223
EC01201=0.0000,2141.5079
EC01202=0.0000,2143.2579
EC01203=0.0000,2144.8552
EC01204=0.0000,2146.1003
EC01205=0.0000,2147.0872
EC01206=0.0000,2148.0658
EC01207=0.0000,2149.2879
EC01208=0.0000,2151.0850
EC01209=0.0000,2153.7379
EC01210=0.0000,2156.7146
EC01211=0.0000,2160.0000
EC01212=0.0000,2160.0000
EC01213=0.0000,2163.2709
EC01214=0.0000,2166.2435
EC01215=0.0000,2168.8988
EC01216=0.0000,2170.6850
EC01217=0.0000,2171.8912
EC01218=0.0000,2172.8520
EC01219=0.0000,2173.8189
EC01220=0.0000,2175.0400
EC01221=0.0000,2176.6318
EC01222=0.0000,2178.3974
EC01223=0.0000,2180.1155
EC01224=0.0000,2181.7171
EC01225=0.0000,2183.2826
EC01226=0.0000,2184.8847
EC01227=0.0000,2186.6022
EC01228=0.0000,2188.3677
EC01229=0.0000,2189.9600
EC01230=0.0000,2191.1815
EC01231=0.0000,2192.1481
EC01232=0.0000,2193.1089
EC01233=0.0000,2194.3149
EC01234=0.0000,2196.1008
EC01235=0.0000,2198.7567
EC01236=0.0000,2201.7290
EC01237=0.0000,2205.0000
EC01238=0.0000,2208.2710
EC01239=0.0000,2211.2433
EC01240=0.0000,2213.8992
EC01241=0.0000,2215.6851
EC01242=0.0000,2216.8911
EC01243=0.0000,2217.8519
EC01244=0.0000,2218.8185
EC01245=0.0000,2220.0400
EC01246=0.0000,2221.6323
EC01247=0.0000,2223.3978
EC01248=0.0000,2225.1153
EC01249=0.0000,2226.7174
EC01250=0.0000,2228.2829
EC01251=0.0000,2229.8845
EC01252=0.0000,2231.6026
EC01253=0.0000,2233.3682
EC01254=0.0000,2234.9600
EC01255=0.0000,2236.1811
EC01256=0.0000,2237.1480
EC01257=0.0000,2238.1088
EC01258=0.0000,2239.3150
EC01259=0.0000,2241.1012
EC01260=0.0000,2243.7565
EC01261=0.0000,2246.7291
EC01262=0.0000,2250.0000
EC01263=0.0000,2253.2709
EC01264=0.0000,2256.2435
EC01265=0.0000,2258.8988
EC01266=0.0000,2260.6850
EC01267=0.0000,2261.8912
EC01268=0.0000,2262.8520
EC01269=0.0000,2263.8189
EC01270=0.0000,2265.0400
EC01271=0.0000,2266.6318
EC01272=0.0000,2268.3974
EC01273=0.0000,2270.1155
EC01274=0.0000,2271.7171
EC01275=0.0000,2273.2826
EC01276=0.0000,2274.8847
EC01277=0.0000,2276.6022
EC01278=0.0000,2278.3677
EC01279=0.0000,2279.9600
EC01280=0.0000,2281.1815
EC01281=0.0000,2282.1481
EC01282=0.0000,2283.1089
EC01283=0.0000,2284.3149
EC01284=0.0000,2286.1008
EC01285=0.0000,2288.7567
EC01286=0.0000,2291.7290
EC01287=0.0000,2295.0000
EC01288=0.0000,2298.2710
EC01289=0.0000,2301.2433
EC01290=0.0000,2303.8992
EC01291=0.0000,2305.6851
EC01292=0.0000,2306.8911
EC01293=0.0000,2307.8519
EC01294=0.0000,2308.8185
EC01295=0.0000,2310.0400
EC01296=0.0000,2311.6323
EC01297=0.0000,2313.3978
EC01298=0.0000,2315.1153
EC01299=0.0000,2316.7174
EC01300=0.0000,2318.2829
EC01301=0.0000,2319.8845
EC01302=0.0000,2321.6026
EC01303=0.0000,2323.3682
EC01304=0.0000,2324.9600
EC01305=0.0000,2326.1811
EC01306=0.0000,2327.1480
EC01307=0.0000,2328.1088
EC01308=0.0000,2329.3150
EC01309=0.0000,2331.1012
EC01310=0.0000,2333.7565
EC01311=0.0000,2336.7291
EC01312=0.0000,2340.0000
EC01313=0.0000,2340.0000
EC01314=0.0000,2343.2709
EC01315=0.0000,2346.2435
EC01316=0.0000,2348.8988
EC01317=0.0000,2350.6850
EC01318=0.0000,2351.8912
EC01319=0.0000,2352.8520
EC01320=0.0000,2353.8189
EC01321=0.0000,2355.0400
EC01322=0.0000,2356.6318
EC01323=0.0000,2358.3974
EC01324=0.0000,2360.1155
EC01325=0.0000,2361.7171
EC01326=0.0000,2363.2826
EC01327=0.0000,2364.8847
EC01328=0.0000,2366.6022
EC01329=0.0000,2368.3677
EC01330=0.0000,2369.9600
EC01331=0.0000,2371.1815
EC01332=0.0000,2372.1481
EC01333=0.0000,2373.1089
EC01334=0.0000,2374.3149
EC01335=0.0000,2376.1008
EC01336=0.0000,2378.7567
EC01337=0.0000,2381.7290
EC01338=0.0000,2385.0000
EC01339=0.0000,2388.2710
EC01340=0.0000,2391.2433
EC01341=0.0000,2393.8992
EC01342=0.0000,2395.6851
EC01343=0.0000,2396.8911
EC01344=0.0000,2397.8519
EC01345=0.0000,2398.8185
EC01346=0.0000,2400.0400
EC01347=0.0000,2401.6323
EC01348=0.0000,2403.3978
EC01349=0.0000,2405.1153
EC01350=0.0000,2406.7174
EC01351=0.0000,2408.2829
EC01352=0.0000,2409.8845
EC01353=0.0000,2411.6026
EC01354=0.0000,2413.3682
EC01355=0.0000,2414.9600
EC01356=0.0000,2416.1811
EC01357=0.0000,2417.1480
EC01358=0.0000,2418.1088
EC01359=0.0000,2419.3150
EC01360=0.0000,2421.1012
EC01361=0.0000,2423.7565
EC01362=0.0000,2426.7291
EC01363=0.0000,2430.0000
EC01364=0.0000,2433.2709
EC01365=0.0000,2436.2435
EC01366=0.0000,2438.8988
EC01367=0.0000,2440.6850
EC01368=0.0000,2441.8912
EC01369=0.0000,2442.8520
EC01370=0.0000,2443.8189
EC01371=0.0000,2445.0400
EC01372=0.0000,2446.6318
EC01373=0.0000,2448.3974
EC01374=0.0000,2450.1155
EC01375=0.0000,2451.7171
EC01376=0.0000,2453.2826
EC01377=0.0000,2454.8847
EC01378=0.0000,2456.6022
EC01379=0.0000,2458.3677
EC01380=0.0000,2459.9600
EC01381=0.0000,2461.1815
EC01382=0.0000,2462.1481
EC01383=0.0000,2463.1089
EC01384=0.0000,2464.3149
EC01385=0.0000,2466.1008
EC01386=0.0000,2468.7567
EC01387=0.0000,2471.7290
EC01388=0.0000,2475.0000
EC01389=0.0000,2478.2710
EC01390=0.0000,2481.2433
EC01391=0.0000,2483.8992
EC01392=0.0000,2485.6851
EC01393=0.0000,2486.8911
EC01394=0.0000,2487.8519
EC01395=0.0000,2488.8185
EC01396=0.0000,2490.0400
EC01397=0.0000,2491.6323
EC01398=0.0000,2493.3978
EC01399=0.0000,2495.1153
EC01400=0.0000,2496.7174
EC01401=0.0000,2498.2829
EC01402=0.0000,2499.8845
EC01403=0.0000,2501.6026
EC01404=0.0000,2503.3682
EC01405=0.0000,2504.9600
EC01406=0.0000,2506.1811
EC01407=0.0000,2507.1480
EC01408=0.0000,2508.1088
EC01409=0.0000,2509.3150
EC01410=0.0000,2511.1012
EC01411=0.0000,2513.7565
EC01412=0.0000,2516.7291
EC01413=0.0000,2520.0000
EC01414=0.0000,2520.0000
EC01415=0.0000,2523.2546
EC01416=0.0000,2526.2211
EC01417=0.0000,2528.8807
EC01418=0.0000,2530.6541
EC01419=0.0000,2531.8420
EC01420=0.0000,2532.7823
EC01421=0.0000,2533.7251
EC01422=0.0000,2534.9190
EC01423=0.0000,2536.5054
EC01424=0.0000,2538.2889
EC01425=0.0000,2540.0438
EC01426=0.0000,2541.6927
EC01427=0.0000,2543.3075
EC01428=0.0000,2544.9564
EC01429=0.0000,2546.7113
EC01430=0.0000,2548.4943
EC01431=0.0000,2550.0807
EC01432=0.0000,2551.2747
EC01433=0.0000,2552.2172
EC01434=0.0000,2553.1579
EC01435=0.0000,2554.3457
EC01436=0.0000,2556.1194
EC01437=0.0000,2558.7787
EC01438=0.0000,2561.7455
EC01439=0.0000,2565.0000
EC01440=0.0000,2568.2545
EC01441=0.0000,2571.2213
EC01442=0.0000,2573.8806
EC01443=0.0000,2575.6543
EC01444=0.0000,2576.8421
EC01445=0.0000,2577.7828
EC01446=0.0000,2578.7253
EC01447=0.0000,2579.9193
EC01448=0.0000,2581.5057
EC01449=0.0000,2583.2887
EC01450=0.0000,2585.0436
EC01451=0.0000,2586.6925
EC01452=0.0000,2588.3073
EC01453=0.0000,2589.9562
EC01454=0.0000,2591.7111
EC01455=0.0000,2593.4946
EC01456=0.0000,2595.0810
EC01457=0.0000,2596.2749
EC01458=0.0000,2597.2177
EC01459=0.0000,2598.1580
EC01460=0.0000,2599.3459
EC01461=0.0000,2601.1193
EC01462=0.0000,2603.7789
EC01463=0.0000,2606.7454
EC01464=0.0000,2610.0000
EC01465=0.0000,2613.2546
EC01466=0.0000,2616.2211
EC01467=0.0000,2618.8807
EC01468=0.0000,2620.6541
EC01469=0.0000,2621.8420
EC01470=0.0000,2622.7823
EC01471=0.0000,2623.7251
EC01472=0.0000,2624.9190
EC01473=0.0000,2626.5054
EC01474=0.0000,2628.2889
EC01475=0.0000,2630.0438
EC01476=0.0000,2631.6927
EC01477=0.0000,2633.3075
EC01478=0.0000,2634.9564
EC01479=0.0000,2636.7113
EC01480=0.0000,2638.4943
EC01481=0.0000,2640.0807
EC01482=0.0000,2641.2747
EC01483=0.0000,2642.2172
EC01484=0.0000,2643.1579
EC01485=0.0000,2644.3457
EC01486=0.0000,2646.1194
EC01487=0.0000,2648.7787
EC01488=0.0000,2651.7455
EC01489=0.0000,2655.0000
EC01490=0.0000,2658.2545
EC01491=0.0000,2661.2213
EC01492=0.0000,2663.8806
EC01493=0.0000,2665.6543
EC01494=0.0000,2666.8421
EC01495=0.0000,2667.7828
EC01496=0.0000,2668.7253
EC01497=0.0000,2669.9193
EC01498=0.0000,2671.5057
EC01499=0.0000,2673.2887
EC01500=0.0000,2675.0436
EC01501=0.0000,2676.6925
EC01502=0.0000,2678.3073
EC01503=0.0000,2679.9562
EC01504=0.0000,2681.7111
EC01505=0.0000,2683.4946
EC01506=0.0000,2685.0810
EC01507=0.0000,2686.2749
EC01508=0.0000,2687.2177
EC01509=0.0000,2688.1580
EC01510=0.0000,2689.3459
EC01511=0.0000,2691.1193
EC01512=0.0000,2693.7789
EC01513=0.0000,2696.7454
EC01514=0.0000,2700.0000
EC01515=0.0000,2700.0000
EC01516=0.0000,2703.2546
EC01517=0.0000,2706.2211
EC01518=0.0000,2708.8807
EC01519=0.0000,2710.6541
EC01520=0.0000,2711.8420
EC01521=0.0000,2712.7823
EC01522=0.0000,2713.7251
EC01523=0.0000,2714.9190
EC01524=0.0000,2716.5054
EC01525=0.0000,2718.2889
EC01526=0.0000,2720.0438
EC01527=0.0000,2721.6927
EC01528=0.0000,2723.3075
EC01529=0.0000,2724.9564
EC01530=0.0000,2726.7113
EC01531=0.0000,2728.4943
EC01532=0.0000,2730.0807
EC01533=0.0000,2731.2747
EC01534=0.0000,2732.2172
EC01535=0.0000,2733.1579
EC01536=0.0000,2734.3457
EC01537=0.0000,2736.1194
EC01538=0.0000,2738.7787
EC01539=0.0000,2741.7455
EC01540=0.0000,2745.0000
EC01541=0.0000,2748.2545
EC01542=0.0000,2751.2213
EC01543=0.0000,2753.8806
EC01544=0.0000,2755.6543
EC01545=0.0000,2756.8421
EC01546=0.0000,2757.7828
EC01547=0.0000,2758.7253
EC01548=0.0000,2759.9193
EC01549=0.0000,2761.5057
EC01550=0.0000,2763.2887
EC01551=0.0000,2765.0436
EC01552=0.0000,2766.6925
EC01553=0.0000,2768.3073
EC01554=0.0000,2769.9562
EC01555=0.0000,2771.7111
EC01556=0.0000,2773.4946
EC01557=0.0000,2775.0810
EC01558=0.0000,2776.2749
EC01559=0.0000,2777.2177
EC01560=0.0000,2778.1580
EC01561=0.0000,2779.3459
EC01562=0.0000,2781.1193
EC01563=0.0000,2783.7789
EC01564=0.0000,2786.7454
EC01565=0.0000,2790.0000
EC01566=0.0000,2793.2546
EC01567=0.0000,2796.2211
EC01568=0.0000,2798.8807
EC01569=0.0000,2800.6541
EC01570=0.0000,2801.8420
EC01571=0.0000,2802.7823
EC01572=0.0000,2803.7251
EC01573=0.0000,2804.9190
EC01574=0.0000,2806.5054
EC01575=0.0000,2808.2889
EC01576=0.0000,2810.0438
EC01577=0.0000,2811.6927
EC01578=0.0000,2813.3075
EC01579=0.0000,2814.9564
EC01580=0.0000,2816.7113
EC01581=0.0000,2818.4943
EC01582=0.0000,2820.0807
EC01583=0.0000,2821.2747
EC01584=0.0000,2822.2172
EC01585=0.0000,2823.1579
EC01586=0.0000,2824.3457
EC01587=0.0000,2826.1194
EC01588=0.0000,2828.7787
EC01589=0.0000,2831.7455
EC01590=0.0000,2835.0000
EC01591=0.0000,2838.2545
EC01592=0.0000,2841.2213
EC01593=0.0000,2843.8806
EC01594=0.0000,2845.6543
EC01595=0.0000,2846.8421
EC01596=0.0000,2847.7828
EC01597=0.0000,2848.7253
EC01598=0.0000,2849.9193
EC01599=0.0000,2851.5057
EC01600=0.0000,2853.2887
EC01601=0.0000,2855.0436
EC01602=0.0000,2856.6925
EC01603=0.0000,2858.3073
EC01604=0.0000,2859.9562
EC01605=0.0000,2861.7111
EC01606=0.0000,2863.4946
EC01607=0.0000,2865.0810
EC01608=0.0000,2866.2749
EC01609=0.0000,2867.2177
EC01610=0.0000,2868.1580
EC01611=0.0000,2869.3459
EC01612=0.0000,2871.1193
EC01613=0.0000,2873.7789
EC01614=0.0000,2876.7454
EC01615=0.0000,2880.0000
EC01616=0.0000,2880.0000
EC01617=0.0000,2883.2359
EC01618=0.0000,2886.1970
EC01619=0.0000,2888.8601
EC01620=0.0000,2890.6197
EC01621=0.0000,2891.7864
EC01622=0.0000,2892.7041
EC01623=0.0000,2893.6200
EC01624=0.0000,2894.7831
EC01625=0.0000,2896.3632
EC01626=0.0000,2898.1666
EC01627=0.0000,2899.9634
EC01628=0.0000,2901.6649
EC01629=0.0000,2903.3352
EC01630=0.0000,2905.0366
EC01631=0.0000,2906.8332
EC01632=0.0000,2908.6370
EC01633=0.0000,2910.2167
EC01634=0.0000,2911.3801
EC01635=0.0000,2912.2959
EC01636=0.0000,2913.2134
EC01637=0.0000,2914.3801
EC01638=0.0000,2916.1402
EC01639=0.0000,2918.8032
EC01640=0.0000,2921.7642
EC01641=0.0000,2925.0000
EC01642=0.0000,2928.2358
EC01643=0.0000,2931.1968
EC01644=0.0000,2933.8598
EC01645=0.0000,2935.6199
EC01646=0.0000,2936.7866
EC01647=0.0000,2937.7041
EC01648=0.0000,2938.6199
EC01649=0.0000,2939.7833
EC01650=0.0000,2941.3630
EC01651=0.0000,2943.1668
EC01652=0.0000,2944.9634
EC01653=0.0000,2946.6648
EC01654=0.0000,2948.3351
EC01655=0.0000,2950.0366
EC01656=0.0000,2951.8334
EC01657=0.0000,2953.6368
EC01658=0.0000,2955.2169
EC01659=0.0000,2956.3800
EC01660=0.0000,2957.2959
EC01661=0.0000,2958.2136
EC01662=0.0000,2959.3803
EC01663=0.0000,2961.1399
EC01664=0.0000,2963.8030
EC01665=0.0000,2966.7641
EC01666=0.0000,2970.0000
EC01667=0.0000,2973.2359
EC01668=0.0000,2976.1970
EC01669=0.0000,2978.8601
EC01670=0.0000,2980.6197
EC01671=0.0000,2981.7864
EC01672=0.0000,2982.7041
EC01673=0.0000,2983.6200
EC01674=0.0000,2984.7831
EC01675=0.0000,2986.3632
EC01676=0.0000,2988.1666
EC01677=0.0000,2989.9634
EC01678=0.0000,2991.6649
EC01679=0.0000,2993.3352
EC01680=0.0000,2995.0366
EC01681=0.0000,2996.8332
EC01682=0.0000,2998.6370
EC01683=0.0000,3000.2167
EC01684=0.0000,3001.3801
EC01685=0.0000,3002.2959
EC01686=0.0000,3003.2134
EC01687=0.0000,3004.3801
EC01688=0.0000,3006.1402
EC01689=0.0000,3008.8032
EC01690=0.0000,3011.7642
EC01691=0.0000,3015.0000
EC01692=0.0000,3018.2358
EC01693=0.0000,3021.1968
EC01694=0.0000,3023.8598
EC01695=0.0000,3025.6199
EC01696=0.0000,3026.7866
EC01697=0.0000,3027.7041
EC01698=0.0000,3028.6199
EC01699=0.0000,3029.7833
EC01700=0.0000,3031.3630
EC01701=0.0000,3033.1668
EC01702=0.0000,3034.9634
EC01703=0.0000,3036.6648
EC01704=0.0000,3038.3351
EC01705=0.0000,3040.0366
EC01706=0.0000,3041.8334
EC01707=0.0000,3043.6368
EC01708=0.0000,3045.2169
EC01709=0.0000,3046.3800
EC01710=0.0000,3047.2959
EC01711=0.0000,3048.2136
EC01712=0.0000,3049.3803
EC01713=0.0000,3051.1399
EC01714=0.0000,3053.8030
EC01715=0.0000,3056.7641
EC01716=0.0000,3060.0000
EC01717=0.0000,3060.0000
EC01718=0.0000,3063.2359
EC01719=0.0000,3066.1970
EC01720=0.0000,3068.8601
EC01721=0.0000,3070.6197
EC01722=0.0000,3071.7864
EC01723=0.0000,3072.7041
EC01724=0.0000,3073.6200
EC01725=0.0000,3074.7831
EC01726=0.0000,3076.3632
EC01727=0.0000,3078.1666
EC01728=0.0000,3079.9634
EC01729=0.0000,3081.6649
EC01730=0.0000,3083.3352
EC01731=0.0000,3085.0366
EC01732=0.0000,3086.8332
EC01733=0.0000,3088.6370
EC01734=0.0000,3090.2167
EC01735=0.0000,3091.3801
EC01736=0.0000,3092.2959
EC01737=0.0000,3093.2134
EC01738=0.0000,3094.3801
EC01739=0.0000,3096.1402
EC01740=0.0000,3098.8032
EC01741=0.0000,3101.7642
EC01742=0.0000,3105.0000
EC01743=0.0000,3108.2358
EC01744=0.0000,3111.1968
EC01745=0.0000,3113.8598
EC01746=0.0000,3115.6199
EC01747=0.0000,3116.7866
EC01748=0.0000,3117.7041
EC01749=0.0000,3118.6199
EC01750=0.0000,3119.7833
EC01751=0.0000,3121.3630
EC01752=0.0000,3123.1668
EC01753=0.0000,3124.9634
EC01754=0.0000,3126.6648
EC01755=0.0000,3128.3351
EC01756=0.0000,3130.0366
EC01757=0.0000,3131.8334
EC01758=0.0000,3133.6368
EC01759=0.0000,3135.2169
EC01760=0.0000,3136.3800
EC01761=0.0000,3137.2959
EC01762=0.0000,3138.2136
EC01763=0.0000,3139.3803
EC01764=0.0000,3141.1399
EC01765=0.0000,3143.8030
EC01766=0.0000,3146.7641
EC01767=0.0000,3150.0000
EC01768=0.0000,3153.2359
EC01769=0.0000,3156.1970
EC01770=0.0000,3158.8601
EC01771=0.0000,3160.6197
EC01772=0.0000,3161.7864
EC01773=0.0000,3162.7041
EC01774=0.0000,3163.6200
EC01775=0.0000,3164.7831
EC01776=0.0000,3166.3632
EC01777=0.0000,3168.1666
EC01778=0.0000,3169.9634
EC01779=0.0000,3171.6649
EC01780=0.0000,3173.3352
EC01781=0.0000,3175.0366
EC01782=0.0000,3176.8332
EC01783=0.0000,3178.6370
EC01784=0.0000,3180.2167
EC01785=0.0000,3181.3801
EC01786=0.0000,3182.2959
EC01787=0.0000,3183.2134
EC01788=0.0000,3184.3801
EC01789=0.0000,3186.1402
EC01790=0.0000,3188.8032
EC01791=0.0000,3191.7642
EC01792=0.0000,3195.0000
EC01793=0.0000,3198.2358
EC01794=0.0000,3201.1968
EC01795=0.0000,3203.8598
EC01796=0.0000,3205.6199
EC01797=0.0000,3206.7866
EC01798=0.0000,3207.7041
EC01799=0.0000,3208.6199
EC01800=0.0000,3209.7833
EC01801=0.0000,3211.3630
EC01802=0.0000,3213.1668
EC01803=0.0000,3214.9634
EC01804=0.0000,3216.6648
EC01805=0.0000,3218.3351
EC01806=0.0000,3220.0366
EC01807=0.0000,3221.8334
EC01808=0.0000,3223.6368
EC01809=0.0000,3225.2169
EC01810=0.0000,3226.3800
EC01811=0.0000,3227.2959
EC01812=0.0000,3228.2136
EC01813=0.0000,3229.3803
EC01814=0.0000,3231.1399
EC01815=0.0000,3233.8030
EC01816=0.0000,3236.7641
EC01817=0.0000,3240.0000
EC01818=0.0000,3240.0000
EC01819=0.0000,3243.2152
EC01820=0.0000,3246.1699
EC01821=0.0000,3248.8371
EC01822=0.0000,3250.5819
EC01823=0.0000,3251.7253
EC01824=0.0000,3252.6169
EC01825=0.0000,3253.5035
EC01826=0.0000,3254.6333
EC01827=0.0000,3256.2063
EC01828=0.0000,3258.0324
EC01829=0.0000,3259.8748
EC01830=0.0000,3261.6343
EC01831=0.0000,3263.3660
EC01832=0.0000,3265.1253
EC01833=0.0000,3266.9678
EC01834=0.0000,3268.7935
EC01835=0.0000,3270.3670
EC01836=0.0000,3271.4965
EC01837=0.0000,3272.3830
EC01838=0.0000,3273.2751
EC01839=0.0000,3274.4183
EC01840=0.0000,3276.1625
EC01841=0.0000,3278.8301
EC01842=0.0000,3281.7846
EC01843=0.0000,3285.0000
EC01844=0.0000,3288.2154
EC01845=0.0000,3291.1699
EC01846=0.0000,3293.8375
EC01847=0.0000,3295.5817
EC01848=0.0000,3296.7249
EC01849=0.0000,3297.6170
EC01850=0.0000,3298.5035
EC01851=0.0000,3299.6330
EC01852=0.0000,3301.2065
EC01853=0.0000,3303.0322
EC01854=0.0000,3304.8747
EC01855=0.0000,3306.6340
EC01856=0.0000,3308.3657
EC01857=0.0000,3310.1252
EC01858=0.0000,3311.9676
EC01859=0.0000,3313.7937
EC01860=0.0000,3315.3667
EC01861=0.0000,3316.4965
EC01862=0.0000,3317.3831
EC01863=0.0000,3318.2747
EC01864=0.0000,3319.4181
EC01865=0.0000,3321.1629
EC01866=0.0000,3323.8301
EC01867=0.0000,3326.7848
EC01868=0.0000,3330.0000
EC01869=0.0000,3333.2152
EC01870=0.0000,3336.1699
EC01871=0.0000,3338.8371
EC01872=0.0000,3340.5819
EC01873=0.0000,3341.7253
EC01874=0.0000,3342.6169
EC01875=0.0000,3343.5035
EC01876=0.0000,3344.6333
EC01877=0.0000,3346.2063
EC01878=0.0000,3348.0324
EC01879=0.0000,3349.8748
EC01880=0.0000,3351.6343
EC01881=0.0000,3353.3660
EC01882=0.0000,3355.1253
EC01883=0.0000,3356.9678
EC01884=0.0000,3358.7935
EC01885=0.0000,3360.3670
EC01886=0.0000,3361.4965
EC01887=0.0000,3362.3830
EC01888=0.0000,3363.2751
EC01889=0.0000,3364.4183
EC01890=0.0000,3366.1625
EC01891=0.0000,3368.8301
EC01892=0.0000,3371.7846
EC01893=0.0000,3375.0000
EC01894=0.0000,3378.2154
EC01895=0.0000,3381.1699
EC01896=0.0000,3383.8375
EC01897=0.0000,3385.5817
EC01898=0.0000,3386.7249
EC01899=0.0000,3387.6170
EC01900=0.0000,3388.5035
EC01901=0.0000,3389.6330
EC01902=0.0000,3391.2065
EC01903=0.0000,3393.0322
EC01904=0.0000,3394.8747
EC01905=0.0000,3396.6340
EC01906=0.0000,3398.3657
EC01907=0.0000,3400.1252
EC01908=0.0000,3401.9676
EC01909=0.0000,3403.7937
EC01910=0.0000,3405.3667
EC01911=0.0000,3406.4965
EC01912=0.0000,3407.3831
EC01913=0.0000,3408.2747
EC01914=0.0000,3409.4181
EC01915=0.0000,3411.1629
EC01916=0.0000,3413.8301
EC01917=0.0000,3416.7848
EC01918=0.0000,3420.0000
EC01919=0.0000,3420.0000
EC01920=0.0000,3423.2152
EC01921=0.0000,3426.1699
EC01922=0.0000,3428.8371
EC01923=0.0000,3430.5819
EC01924=0.0000,3431.7253
EC01925=0.0000,3432.6169
EC01926=0.0000,3433.5035
EC01927=0.0000,3434.6333
EC01928=0.0000,3436.2063
EC01929=0.0000,3438.0324
EC01930=0.0000,3439.8748
EC01931=0.0000,3441.6343
EC01932=0.0000,3443.3660
EC01933=0.0000,3445.1253
EC01934=0.0000,3446.9678
EC01935=0.0000,3448.7935
EC01936=0.0000,3450.3670
EC01937=0.0000,3451.4965
EC01938=0.0000,3452.3830
EC01939=0.0000,3453.2751
EC01940=0.0000,3454.4183
EC01941=0.0000,3456.1625
EC01942=0.0000,3458.8301
EC01943=0.0000,3461.7846
EC01944=0.0000,3465.0000
EC01945=0.0000,3468.2154
EC01946=0.0000,3471.1699
EC01947=0.0000,3473.8375
EC01948=0.0000,3475.5817
EC01949=0.0000,3476.7249
EC01950=0.0000,3477.6170
EC01951=0.0000,3478.5035
EC01952=0.0000,3479.6330
EC01953=0.0000,3481.2065
EC01954=0.0000,3483.0322
EC01955=0.0000,3484.8747
EC01956=0.0000,3486.6340
EC01957=0.0000,3488.3657
EC01958=0.0000,3490.1252
EC01959=0.0000,3491.9676
EC01960=0.0000,3493.7937
EC01961=0.0000,3495.3667
EC01962=0.0000,3496.4965
EC01963=0.0000,3497.3831
EC01964=0.0000,3498.2747
EC01965=0.0000,3499.4181
EC01966=0.0000,3501.1629
EC01967=0.0000,3503.8301
EC01968=0.0000,3506.7848
EC01969=0.0000,3510.0000
EC01970=0.0000,3513.2152
EC01971=0.0000,3516.1699
EC01972=0.0000,3518.8371
EC01973=0.0000,3520.5819
EC01974=0.0000,3521.7253
EC01975=0.0000,3522.6169
EC01976=0.0000,3523.5035
EC01977=0.0000,3524.6333
EC01978=0.0000,3526.2063
EC01979=0.0000,3528.0324
EC01980=0.0000,3529.8748
EC01981=0.0000,3531.6343
EC01982=0.0000,3533.3660
EC01983=0.0000,3535.1253
EC01984=0.0000,3536.9678
EC01985=0.0000,3538.7935
EC01986=0.0000,3540.3670
EC01987=0.0000,3541.4965
EC01988=0.0000,3542.3830
EC01989=0.0000,3543.2751
EC01990=0.0000,3544.4183
EC01991=0.0000,3546.1625
EC01992=0.0000,3548.8301
EC01993=0.0000,3551.7846
EC01994=0.0000,3555.0000
EC01995=0.0000,3558.2154
EC01996=0.0000,3561.1699
EC01997=0.0000,3563.8375
EC01998=0.0000,3565.5817
EC01999=0.0000,3566.7249
//INST
///DATE 2022/04/08 11:28
///COMM
///ATTR SC,RW,RJ
////FRAME USER 2
///GROUP1 RB1
///GROUP2 ST1
NOP
SPEED V=20.0
SMOVL C00000 +MOVJ EC00000
ARCON
SMOVL C00001 +MOVJ EC00001
SPEED V=19.0
SMOVL C00002 +MOVJ EC00002
SPEED V=18.0
SMOVL C00003 +MOVJ EC00003
SPEED V=17.0
SMOVL C00004 +MOVJ EC00004
SPEED V=16.0
SMOVL C00005 +MOVJ EC00005
SPEED V=15.0
SMOVL C00006 +MOVJ EC00006
SPEED V=14.0
SMOVL C00007 +MOVJ EC00007
SPEED V=13.0
SMOVL C00008 +MOVJ EC00008
SPEED V=12.0
SMOVL C00009 +MOVJ EC00009
SPEED V=11.0
SMOVL C00010 +MOVJ EC00010
SPEED V=10.0
SMOVL C00011 +MOVJ EC00011
SMOVL C00012 +MOVJ EC00012
SMOVL C00013 +MOVJ EC00013
SMOVL C00014 +MOVJ EC00014
SMOVL C00015 +MOVJ EC00015
SMOVL C00016 +MOVJ EC00016
SMOVL C00017 +MOVJ EC00017
SMOVL C00018 +MOVJ EC00018
SMOVL C00019 +MOVJ EC00019
SMOVL C00020 +MOVJ EC00020
SMOVL C00021 +MOVJ EC00021
SMOVL C00022 +MOVJ EC00022
SMOVL C00023 +MOVJ EC00023
SMOVL C00024 +MOVJ EC00024
SMOVL C00025 +MOVJ EC00025
SMOVL C00026 +MOVJ EC00026
SMOVL C00027 +MOVJ EC00027
SMOVL C00028 +MOVJ EC00028
SMOVL C00029 +MOVJ EC00029
SMOVL C00030 +MOVJ EC00030
SMOVL C00031 +MOVJ EC00031
SMOVL C00032 +MOVJ EC00032
SMOVL C00033 +MOVJ EC00033
SMOVL C00034 +MOVJ EC00034
SMOVL C00035 +MOVJ EC00035
SMOVL C00036 +MOVJ EC00036
SMOVL C00037 +MOVJ EC00037
SMOVL C00038 +MOVJ EC00038
SMOVL C00039 +MOVJ EC00039
SMOVL C00040 +MOVJ EC00040
SMOVL C00041 +MOVJ EC00041
SMOVL C00042 +MOVJ EC00042
SMOVL C00043 +MOVJ EC00043
SMOVL C00044 +MOVJ EC00044
SMOVL C00045 +MOVJ EC00045
SMOVL C00046 +MOVJ EC00046
SMOVL C00047 +MOVJ EC00047
SMOVL C00048 +MOVJ EC00048
SMOVL C00049 +MOVJ EC00049
SMOVL C00050 +MOVJ EC00050
SMOVL C00051 +MOVJ EC00051
SMOVL C00052 +MOVJ EC00052
SMOVL C00053 +MOVJ EC00053
SMOVL C00054 +MOVJ EC00054
SMOVL C00055 +MOVJ EC00055
SMOVL C00056 +MOVJ EC00056
SMOVL C00057 +MOVJ EC00057
SMOVL C00058 +MOVJ EC00058
SMOVL C00059 +MOVJ EC00059
SMOVL C00060 +MOVJ EC00060
SMOVL C00061 +MOVJ EC00061
SMOVL C00062 +MOVJ EC00062
SMOVL C00063 +MOVJ EC00063
SMOVL C00064 +MOVJ EC00064
SMOVL C00065 +MOVJ EC00065
SMOVL C00066 +MOVJ EC00066
SMOVL C00067 +MOVJ EC00067
SMOVL C00068 +MOVJ EC00068
SMOVL C00069 +MOVJ EC00069
SMOVL C00070 +MOVJ EC00070
SMOVL C00071 +MOVJ EC00071
SMOVL C00072 +MOVJ EC00072
SMOVL C00073 +MOVJ EC00073
SMOVL C00074 +MOVJ EC00074
SMOVL C00075 +MOVJ EC00075
SMOVL C00076 +MOVJ EC00076
SMOVL C00077 +MOVJ EC00077
SMOVL C00078 +MOVJ EC00078
SMOVL C00079 +MOVJ EC00079
SMOVL C00080 +MOVJ EC00080
SMOVL C00081 +MOVJ EC00081
SMOVL C00082 +MOVJ EC00082
SMOVL C00083 +MOVJ EC00083
SMOVL C00084 +MOVJ EC00084
SMOVL C00085 +MOVJ EC00085
SMOVL C00086 +MOVJ EC00086
SMOVL C00087 +MOVJ EC00087
SMOVL C00088 +MOVJ EC00088
SMOVL C00089 +MOVJ EC00089
SMOVL C00090 +MOVJ EC00090
SMOVL C00091 +MOVJ EC00091
SMOVL C00092 +MOVJ EC00092
SMOVL C00093 +MOVJ EC00093
SMOVL C00094 +MOVJ EC00094
SMOVL C00095 +MOVJ EC00095
SMOVL C00096 +MOVJ EC00096
SMOVL C00097 +MOVJ EC00097
SMOVL C00098 +MOVJ EC00098
SMOVL C00099 +MOVJ EC00099
SMOVL C00100 +MOVJ EC00100
SMOVL C00101 +MOVJ EC00101
SMOVL C00102 +MOVJ EC00102
SMOVL C00103 +MOVJ EC00103
SMOVL C00104 +MOVJ EC00104
SMOVL C00105 +MOVJ EC00105
SMOVL C00106 +MOVJ EC00106
SMOVL C00107 +MOVJ EC00107
SMOVL C00108 +MOVJ EC00108
SMOVL C00109 +MOVJ EC00109
SMOVL C00110 +MOVJ EC00110
SMOVL C00111 +MOVJ EC00111
SMOVL C00112 +MOVJ EC00112
SMOVL C00113 +MOVJ EC00113
SMOVL C00114 +MOVJ EC00114
SMOVL C00115 +MOVJ EC00115
SMOVL C00116 +MOVJ EC00116
SMOVL C00117 +MOVJ EC00117
SMOVL C00118 +MOVJ EC00118
SMOVL C00119 +MOVJ EC00119
SMOVL C00120 +MOVJ EC00120
SMOVL C00121 +MOVJ EC00121
SMOVL C00122 +MOVJ EC00122
SMOVL C00123 +MOVJ EC00123
SMOVL C00124 +MOVJ EC00124
SMOVL C00125 +MOVJ EC00125
SMOVL C00126 +MOVJ EC00126
SMOVL C00127 +MOVJ EC00127
SMOVL C00128 +MOVJ EC00128
SMOVL C00129 +MOVJ EC00129
SMOVL C00130 +MOVJ EC00130
SMOVL C00131 +MOVJ EC00131
SMOVL C00132 +MOVJ EC00132
SMOVL C00133 +MOVJ EC00133
SMOVL C00134 +MOVJ EC00134
SMOVL C00135 +MOVJ EC00135
SMOVL C00136 +MOVJ EC00136
SMOVL C00137 +MOVJ EC00137
SMOVL C00138 +MOVJ EC00138
SMOVL C00139 +MOVJ EC00139
SMOVL C00140 +MOVJ EC00140
SMOVL C00141 +MOVJ EC00141
SMOVL C00142 +MOVJ EC00142
SMOVL C00143 +MOVJ EC00143
SMOVL C00144 +MOVJ EC00144
SMOVL C00145 +MOVJ EC00145
SMOVL C00146 +MOVJ EC00146
SMOVL C00147 +MOVJ EC00147
SMOVL C00148 +MOVJ EC00148
SMOVL C00149 +MOVJ EC00149
SMOVL C00150 +MOVJ EC00150
SMOVL C00151 +MOVJ EC00151
SMOVL C00152 +MOVJ EC00152
SMOVL C00153 +MOVJ EC00153
SMOVL C00154 +MOVJ EC00154
SMOVL C00155 +MOVJ EC00155
SMOVL C00156 +MOVJ EC00156
SMOVL C00157 +MOVJ EC00157
SMOVL C00158 +MOVJ EC00158
SMOVL C00159 +MOVJ EC00159
SMOVL C00160 +MOVJ EC00160
SMOVL C00161 +MOVJ EC00161
SMOVL C00162 +MOVJ EC00162
SMOVL C00163 +MOVJ EC00163
SMOVL C00164 +MOVJ EC00164
SMOVL C00165 +MOVJ EC00165
SMOVL C00166 +MOVJ EC00166
SMOVL C00167 +MOVJ EC00167
SMOVL C00168 +MOVJ EC00168
SMOVL C00169 +MOVJ EC00169
SMOVL C00170 +MOVJ EC00170
SMOVL C00171 +MOVJ EC00171
SMOVL C00172 +MOVJ EC00172
SMOVL C00173 +MOVJ EC00173
SMOVL C00174 +MOVJ EC00174
SMOVL C00175 +MOVJ EC00175
SMOVL C00176 +MOVJ EC00176
SMOVL C00177 +MOVJ EC00177
SMOVL C00178 +MOVJ EC00178
SMOVL C00179 +MOVJ EC00179
SMOVL C00180 +MOVJ EC00180
SMOVL C00181 +MOVJ EC00181
SMOVL C00182 +MOVJ EC00182
SMOVL C00183 +MOVJ EC00183
SMOVL C00184 +MOVJ EC00184
SMOVL C00185 +MOVJ EC00185
SMOVL C00186 +MOVJ EC00186
SMOVL C00187 +MOVJ EC00187
SMOVL C00188 +MOVJ EC00188
SMOVL C00189 +MOVJ EC00189
SMOVL C00190 +MOVJ EC00190
SMOVL C00191 +MOVJ EC00191
SMOVL C00192 +MOVJ EC00192
SMOVL C00193 +MOVJ EC00193
SMOVL C00194 +MOVJ EC00194
SMOVL C00195 +MOVJ EC00195
SMOVL C00196 +MOVJ EC00196
SMOVL C00197 +MOVJ EC00197
SMOVL C00198 +MOVJ EC00198
SMOVL C00199 +MOVJ EC00199
SMOVL C00200 +MOVJ EC00200
SMOVL C00201 +MOVJ EC00201
SMOVL C00202 +MOVJ EC00202
SMOVL C00203 +MOVJ EC00203
SMOVL C00204 +MOVJ EC00204
SMOVL C00205 +MOVJ EC00205
SMOVL C00206 +MOVJ EC00206
SMOVL C00207 +MOVJ EC00207
SMOVL C00208 +MOVJ EC00208
SMOVL C00209 +MOVJ EC00209
SMOVL C00210 +MOVJ EC00210
SMOVL C00211 +MOVJ EC00211
SMOVL C00212 +MOVJ EC00212
SMOVL C00213 +MOVJ EC00213
SMOVL C00214 +MOVJ EC00214
SMOVL C00215 +MOVJ EC00215
SMOVL C00216 +MOVJ EC00216
SMOVL C00217 +MOVJ EC00217
SMOVL C00218 +MOVJ EC00218
SMOVL C00219 +MOVJ EC00219
SMOVL C00220 +MOVJ EC00220
SMOVL C00221 +MOVJ EC00221
SMOVL C00222 +MOVJ EC00222
SMOVL C00223 +MOVJ EC00223
SMOVL C00224 +MOVJ EC00224
SMOVL C00225 +MOVJ EC00225
SMOVL C00226 +MOVJ EC00226
SMOVL C00227 +MOVJ EC00227
SMOVL C00228 +MOVJ EC00228
SMOVL C00229 +MOVJ EC00229
SMOVL C00230 +MOVJ EC00230
SMOVL C00231 +MOVJ EC00231
SMOVL C00232 +MOVJ EC00232
SMOVL C00233 +MOVJ EC00233
SMOVL C00234 +MOVJ EC00234
SMOVL C00235 +MOVJ EC00235
SMOVL C00236 +MOVJ EC00236
SMOVL C00237 +MOVJ EC00237
SMOVL C00238 +MOVJ EC00238
SMOVL C00239 +MOVJ EC00239
SMOVL C00240 +MOVJ EC00240
SMOVL C00241 +MOVJ EC00241
SMOVL C00242 +MOVJ EC00242
SMOVL C00243 +MOVJ EC00243
SMOVL C00244 +MOVJ EC00244
SMOVL C00245 +MOVJ EC00245
SMOVL C00246 +MOVJ EC00246
SMOVL C00247 +MOVJ EC00247
SMOVL C00248 +MOVJ EC00248
SMOVL C00249 +MOVJ EC00249
SMOVL C00250 +MOVJ EC00250
SMOVL C00251 +MOVJ EC00251
SMOVL C00252 +MOVJ EC00252
SMOVL C00253 +MOVJ EC00253
SMOVL C00254 +MOVJ EC00254
SMOVL C00255 +MOVJ EC00255
SMOVL C00256 +MOVJ EC00256
SMOVL C00257 +MOVJ EC00257
SMOVL C00258 +MOVJ EC00258
SMOVL C00259 +MOVJ EC00259
SMOVL C00260 +MOVJ EC00260
SMOVL C00261 +MOVJ EC00261
SMOVL C00262 +MOVJ EC00262
SMOVL C00263 +MOVJ EC00263
SMOVL C00264 +MOVJ EC00264
SMOVL C00265 +MOVJ EC00265
SMOVL C00266 +MOVJ EC00266
SMOVL C00267 +MOVJ EC00267
SMOVL C00268 +MOVJ EC00268
SMOVL C00269 +MOVJ EC00269
SMOVL C00270 +MOVJ EC00270
SMOVL C00271 +MOVJ EC00271
SMOVL C00272 +MOVJ EC00272
SMOVL C00273 +MOVJ EC00273
SMOVL C00274 +MOVJ EC00274
SMOVL C00275 +MOVJ EC00275
SMOVL C00276 +MOVJ EC00276
SMOVL C00277 +MOVJ EC00277
SMOVL C00278 +MOVJ EC00278
SMOVL C00279 +MOVJ EC00279
SMOVL C00280 +MOVJ EC00280
SMOVL C00281 +MOVJ EC00281
SMOVL C00282 +MOVJ EC00282
SMOVL C00283 +MOVJ EC00283
SMOVL C00284 +MOVJ EC00284
SMOVL C00285 +MOVJ EC00285
SMOVL C00286 +MOVJ EC00286
SMOVL C00287 +MOVJ EC00287
SMOVL C00288 +MOVJ EC00288
SMOVL C00289 +MOVJ EC00289
SMOVL C00290 +MOVJ EC00290
SMOVL C00291 +MOVJ EC00291
SMOVL C00292 +MOVJ EC00292
SMOVL C00293 +MOVJ EC00293
SMOVL C00294 +MOVJ EC00294
SMOVL C00295 +MOVJ EC00295
SMOVL C00296 +MOVJ EC00296
SMOVL C00297 +MOVJ EC00297
SMOVL C00298 +MOVJ EC00298
SMOVL C00299 +MOVJ EC00299
SMOVL C00300 +MOVJ EC00300
SMOVL C00301 +MOVJ EC00301
SMOVL C00302 +MOVJ EC00302
SMOVL C00303 +MOVJ EC00303
SMOVL C00304 +MOVJ EC00304
SMOVL C00305 +MOVJ EC00305
SMOVL C00306 +MOVJ EC00306
SMOVL C00307 +MOVJ EC00307
SMOVL C00308 +MOVJ EC00308
SMOVL C00309 +MOVJ EC00309
SMOVL C00310 +MOVJ EC00310
SMOVL C00311 +MOVJ EC00311
SMOVL C00312 +MOVJ EC00312
SMOVL C00313 +MOVJ EC00313
SMOVL C00314 +MOVJ EC00314
SMOVL C00315 +MOVJ EC00315
SMOVL C00316 +MOVJ EC00316
SMOVL C00317 +MOVJ EC00317
SMOVL C00318 +MOVJ EC00318
SMOVL C00319 +MOVJ EC00319
SMOVL C00320 +MOVJ EC00320
SMOVL C00321 +MOVJ EC00321
SMOVL C00322 +MOVJ EC00322
SMOVL C00323 +MOVJ EC00323
SMOVL C00324 +MOVJ EC00324
SMOVL C00325 +MOVJ EC00325
SMOVL C00326 +MOVJ EC00326
SMOVL C00327 +MOVJ EC00327
SMOVL C00328 +MOVJ EC00328
SMOVL C00329 +MOVJ EC00329
SMOVL C00330 +MOVJ EC00330
SMOVL C00331 +MOVJ EC00331
SMOVL C00332 +MOVJ EC00332
SMOVL C00333 +MOVJ EC00333
SMOVL C00334 +MOVJ EC00334
SMOVL C00335 +MOVJ EC00335
SMOVL C00336 +MOVJ EC00336
SMOVL C00337 +MOVJ EC00337
SMOVL C00338 +MOVJ EC00338
SMOVL C00339 +MOVJ EC00339
SMOVL C00340 +MOVJ EC00340
SMOVL C00341 +MOVJ EC00341
SMOVL C00342 +MOVJ EC00342
SMOVL C00343 +MOVJ EC00343
SMOVL C00344 +MOVJ EC00344
SMOVL C00345 +MOVJ EC00345
SMOVL C00346 +MOVJ EC00346
SMOVL C00347 +MOVJ EC00347
SMOVL C00348 +MOVJ EC00348
SMOVL C00349 +MOVJ EC00349
SMOVL C00350 +MOVJ EC00350
SMOVL C00351 +MOVJ EC00351
SMOVL C00352 +MOVJ EC00352
SMOVL C00353 +MOVJ EC00353
SMOVL C00354 +MOVJ EC00354
SMOVL C00355 +MOVJ EC00355
SMOVL C00356 +MOVJ EC00356
SMOVL C00357 +MOVJ EC00357
SMOVL C00358 +MOVJ EC00358
SMOVL C00359 +MOVJ EC00359
SMOVL C00360 +MOVJ EC00360
SMOVL C00361 +MOVJ EC00361
SMOVL C00362 +MOVJ EC00362
SMOVL C00363 +MOVJ EC00363
SMOVL C00364 +MOVJ EC00364
SMOVL C00365 +MOVJ EC00365
SMOVL C00366 +MOVJ EC00366
SMOVL C00367 +MOVJ EC00367
SMOVL C00368 +MOVJ EC00368
SMOVL C00369 +MOVJ EC00369
SMOVL C00370 +MOVJ EC00370
SMOVL C00371 +MOVJ EC00371
SMOVL C00372 +MOVJ EC00372
SMOVL C00373 +MOVJ EC00373
SMOVL C00374 +MOVJ EC00374
SMOVL C00375 +MOVJ EC00375
SMOVL C00376 +MOVJ EC00376
SMOVL C00377 +MOVJ EC00377
SMOVL C00378 +MOVJ EC00378
SMOVL C00379 +MOVJ EC00379
SMOVL C00380 +MOVJ EC00380
SMOVL C00381 +MOVJ EC00381
SMOVL C00382 +MOVJ EC00382
SMOVL C00383 +MOVJ EC00383
SMOVL C00384 +MOVJ EC00384
SMOVL C00385 +MOVJ EC00385
SMOVL C00386 +MOVJ EC00386
SMOVL C00387 +MOVJ EC00387
SMOVL C00388 +MOVJ EC00388
SMOVL C00389 +MOVJ EC00389
SMOVL C00390 +MOVJ EC00390
SMOVL C00391 +MOVJ EC00391
SMOVL C00392 +MOVJ EC00392
SMOVL C00393 +MOVJ EC00393
SMOVL C00394 +MOVJ EC00394
SMOVL C00395 +MOVJ EC00395
SMOVL C00396 +MOVJ EC00396
SMOVL C00397 +MOVJ EC00397
SMOVL C00398 +MOVJ EC00398
SMOVL C00399 +MOVJ EC00399
SMOVL C00400 +MOVJ EC00400
SMOVL C00401 +MOVJ EC00401
SMOVL C00402 +MOVJ EC00402
SMOVL C00403 +MOVJ EC00403
SMOVL C00404 +MOVJ EC00404
SMOVL C00405 +MOVJ EC00405
SMOVL C00406 +MOVJ EC00406
SMOVL C00407 +MOVJ EC00407
SMOVL C00408 +MOVJ EC00408
SMOVL C00409 +MOVJ EC00409
SMOVL C00410 +MOVJ EC00410
SMOVL C00411 +MOVJ EC00411
SMOVL C00412 +MOVJ EC00412
SMOVL C00413 +MOVJ EC00413
SMOVL C00414 +MOVJ EC00414
SMOVL C00415 +MOVJ EC00415
SMOVL C00416 +MOVJ EC00416
SMOVL C00417 +MOVJ EC00417
SMOVL C00418 +MOVJ EC00418
SMOVL C00419 +MOVJ EC00419
SMOVL C00420 +MOVJ EC00420
SMOVL C00421 +MOVJ EC00421
SMOVL C00422 +MOVJ EC00422
SMOVL C00423 +MOVJ EC00423
SMOVL C00424 +MOVJ EC00424
SMOVL C00425 +MOVJ EC00425
SMOVL C00426 +MOVJ EC00426
SMOVL C00427 +MOVJ EC00427
SMOVL C00428 +MOVJ EC00428
SMOVL C00429 +MOVJ EC00429
SMOVL C00430 +MOVJ EC00430
SMOVL C00431 +MOVJ EC00431
SMOVL C00432 +MOVJ EC00432
SMOVL C00433 +MOVJ EC00433
SMOVL C00434 +MOVJ EC00434
SMOVL C00435 +MOVJ EC00435
SMOVL C00436 +MOVJ EC00436
SMOVL C00437 +MOVJ EC00437
SMOVL C00438 +MOVJ EC00438
SMOVL C00439 +MOVJ EC00439
SMOVL C00440 +MOVJ EC00440
SMOVL C00441 +MOVJ EC00441
SMOVL C00442 +MOVJ EC00442
SMOVL C00443 +MOVJ EC00443
SMOVL C00444 +MOVJ EC00444
SMOVL C00445 +MOVJ EC00445
SMOVL C00446 +MOVJ EC00446
SMOVL C00447 +MOVJ EC00447
SMOVL C00448 +MOVJ EC00448
SMOVL C00449 +MOVJ EC00449
SMOVL C00450 +MOVJ EC00450
SMOVL C00451 +MOVJ EC00451
SMOVL C00452 +MOVJ EC00452
SMOVL C00453 +MOVJ EC00453
SMOVL C00454 +MOVJ EC00454
SMOVL C00455 +MOVJ EC00455
SMOVL C00456 +MOVJ EC00456
SMOVL C00457 +MOVJ EC00457
SMOVL C00458 +MOVJ EC00458
SMOVL C00459 +MOVJ EC00459
SMOVL C00460 +MOVJ EC00460
SMOVL C00461 +MOVJ EC00461
SMOVL C00462 +MOVJ EC00462
SMOVL C00463 +MOVJ EC00463
SMOVL C00464 +MOVJ EC00464
SMOVL C00465 +MOVJ EC00465
SMOVL C00466 +MOVJ EC00466
SMOVL C00467 +MOVJ EC00467
SMOVL C00468 +MOVJ EC00468
SMOVL C00469 +MOVJ EC00469
SMOVL C00470 +MOVJ EC00470
SMOVL C00471 +MOVJ EC00471
SMOVL C00472 +MOVJ EC00472
SMOVL C00473 +MOVJ EC00473
SMOVL C00474 +MOVJ EC00474
SMOVL C00475 +MOVJ EC00475
SMOVL C00476 +MOVJ EC00476
SMOVL C00477 +MOVJ EC00477
SMOVL C00478 +MOVJ EC00478
SMOVL C00479 +MOVJ EC00479
SMOVL C00480 +MOVJ EC00480
SMOVL C00481 +MOVJ EC00481
SMOVL C00482 +MOVJ EC00482
SMOVL C00483 +MOVJ EC00483
SMOVL C00484 +MOVJ EC00484
SMOVL C00485 +MOVJ EC00485
SMOVL C00486 +MOVJ EC00486
SMOVL C00487 +MOVJ EC00487
SMOVL C00488 +MOVJ EC00488
SMOVL C00489 +MOVJ EC00489
SMOVL C00490 +MOVJ EC00490
SMOVL C00491 +MOVJ EC00491
SMOVL C00492 +MOVJ EC00492
SMOVL C00493 +MOVJ EC00493
SMOVL C00494 +MOVJ EC00494
SMOVL C00495 +MOVJ EC00495
SMOVL C00496 +MOVJ EC00496
SMOVL C00497 +MOVJ EC00497
SMOVL C00498 +MOVJ EC00498
SMOVL C00499 +MOVJ EC00499
SMOVL C00500 +MOVJ EC00500
SMOVL C00501 +MOVJ EC00501
SMOVL C00502 +MOVJ EC00502
SMOVL C00503 +MOVJ EC00503
SMOVL C00504 +MOVJ EC00504
SMOVL C00505 +MOVJ EC00505
SMOVL C00506 +MOVJ EC00506
SMOVL C00507 +MOVJ EC00507
SMOVL C00508 +MOVJ EC00508
SMOVL C00509 +MOVJ EC00509
SMOVL C00510 +MOVJ EC00510
SMOVL C00511 +MOVJ EC00511
SMOVL C00512 +MOVJ EC00512
SMOVL C00513 +MOVJ EC00513
SMOVL C00514 +MOVJ EC00514
SMOVL C00515 +MOVJ EC00515
SMOVL C00516 +MOVJ EC00516
SMOVL C00517 +MOVJ EC00517
SMOVL C00518 +MOVJ EC00518
SMOVL C00519 +MOVJ EC00519
SMOVL C00520 +MOVJ EC00520
SMOVL C00521 +MOVJ EC00521
SMOVL C00522 +MOVJ EC00522
SMOVL C00523 +MOVJ EC00523
SMOVL C00524 +MOVJ EC00524
SMOVL C00525 +MOVJ EC00525
SMOVL C00526 +MOVJ EC00526
SMOVL C00527 +MOVJ EC00527
SMOVL C00528 +MOVJ EC00528
SMOVL C00529 +MOVJ EC00529
SMOVL C00530 +MOVJ EC00530
SMOVL C00531 +MOVJ EC00531
SMOVL C00532 +MOVJ EC00532
SMOVL C00533 +MOVJ EC00533
SMOVL C00534 +MOVJ EC00534
SMOVL C00535 +MOVJ EC00535
SMOVL C00536 +MOVJ EC00536
SMOVL C00537 +MOVJ EC00537
SMOVL C00538 +MOVJ EC00538
SMOVL C00539 +MOVJ EC00539
SMOVL C00540 +MOVJ EC00540
SMOVL C00541 +MOVJ EC00541
SMOVL C00542 +MOVJ EC00542
SMOVL C00543 +MOVJ EC00543
SMOVL C00544 +MOVJ EC00544
SMOVL C00545 +MOVJ EC00545
SMOVL C00546 +MOVJ EC00546
SMOVL C00547 +MOVJ EC00547
SMOVL C00548 +MOVJ EC00548
SMOVL C00549 +MOVJ EC00549
SMOVL C00550 +MOVJ EC00550
SMOVL C00551 +MOVJ EC00551
SMOVL C00552 +MOVJ EC00552
SMOVL C00553 +MOVJ EC00553
SMOVL C00554 +MOVJ EC00554
SMOVL C00555 +MOVJ EC00555
SMOVL C00556 +MOVJ EC00556
SMOVL C00557 +MOVJ EC00557
SMOVL C00558 +MOVJ EC00558
SMOVL C00559 +MOVJ EC00559
SMOVL C00560 +MOVJ EC00560
SMOVL C00561 +MOVJ EC00561
SMOVL C00562 +MOVJ EC00562
SMOVL C00563 +MOVJ EC00563
SMOVL C00564 +MOVJ EC00564
SMOVL C00565 +MOVJ EC00565
SMOVL C00566 +MOVJ EC00566
SMOVL C00567 +MOVJ EC00567
SMOVL C00568 +MOVJ EC00568
SMOVL C00569 +MOVJ EC00569
SMOVL C00570 +MOVJ EC00570
SMOVL C00571 +MOVJ EC00571
SMOVL C00572 +MOVJ EC00572
SMOVL C00573 +MOVJ EC00573
SMOVL C00574 +MOVJ EC00574
SMOVL C00575 +MOVJ EC00575
SMOVL C00576 +MOVJ EC00576
SMOVL C00577 +MOVJ EC00577
SMOVL C00578 +MOVJ EC00578
SMOVL C00579 +MOVJ EC00579
SMOVL C00580 +MOVJ EC00580
SMOVL C00581 +MOVJ EC00581
SMOVL C00582 +MOVJ EC00582
SMOVL C00583 +MOVJ EC00583
SMOVL C00584 +MOVJ EC00584
SMOVL C00585 +MOVJ EC00585
SMOVL C00586 +MOVJ EC00586
SMOVL C00587 +MOVJ EC00587
SMOVL C00588 +MOVJ EC00588
SMOVL C00589 +MOVJ EC00589
SMOVL C00590 +MOVJ EC00590
SMOVL C00591 +MOVJ EC00591
SMOVL C00592 +MOVJ EC00592
SMOVL C00593 +MOVJ EC00593
SMOVL C00594 +MOVJ EC00594
SMOVL C00595 +MOVJ EC00595
SMOVL C00596 +MOVJ EC00596
SMOVL C00597 +MOVJ EC00597
SMOVL C00598 +MOVJ EC00598
SMOVL C00599 +MOVJ EC00599
SMOVL C00600 +MOVJ EC00600
SMOVL C00601 +MOVJ EC00601
SMOVL C00602 +MOVJ EC00602
SMOVL C00603 +MOVJ EC00603
SMOVL C00604 +MOVJ EC00604
SMOVL C00605 +MOVJ EC00605
SMOVL C00606 +MOVJ EC00606
SMOVL C00607 +MOVJ EC00607
SMOVL C00608 +MOVJ EC00608
SMOVL C00609 +MOVJ EC00609
SMOVL C00610 +MOVJ EC00610
SMOVL C00611 +MOVJ EC00611
SMOVL C00612 +MOVJ EC00612
SMOVL C00613 +MOVJ EC00613
SMOVL C00614 +MOVJ EC00614
SMOVL C00615 +MOVJ EC00615
SMOVL C00616 +MOVJ EC00616
SMOVL C00617 +MOVJ EC00617
SMOVL C00618 +MOVJ EC00618
SMOVL C00619 +MOVJ EC00619
SMOVL C00620 +MOVJ EC00620
SMOVL C00621 +MOVJ EC00621
SMOVL C00622 +MOVJ EC00622
SMOVL C00623 +MOVJ EC00623
SMOVL C00624 +MOVJ EC00624
SMOVL C00625 +MOVJ EC00625
SMOVL C00626 +MOVJ EC00626
SMOVL C00627 +MOVJ EC00627
SMOVL C00628 +MOVJ EC00628
SMOVL C00629 +MOVJ EC00629
SMOVL C00630 +MOVJ EC00630
SMOVL C00631 +MOVJ EC00631
SMOVL C00632 +MOVJ EC00632
SMOVL C00633 +MOVJ EC00633
SMOVL C00634 +MOVJ EC00634
SMOVL C00635 +MOVJ EC00635
SMOVL C00636 +MOVJ EC00636
SMOVL C00637 +MOVJ EC00637
SMOVL C00638 +MOVJ EC00638
SMOVL C00639 +MOVJ EC00639
SMOVL C00640 +MOVJ EC00640
SMOVL C00641 +MOVJ EC00641
SMOVL C00642 +MOVJ EC00642
SMOVL C00643 +MOVJ EC00643
SMOVL C00644 +MOVJ EC00644
SMOVL C00645 +MOVJ EC00645
SMOVL C00646 +MOVJ EC00646
SMOVL C00647 +MOVJ EC00647
SMOVL C00648 +MOVJ EC00648
SMOVL C00649 +MOVJ EC00649
SMOVL C00650 +MOVJ EC00650
SMOVL C00651 +MOVJ EC00651
SMOVL C00652 +MOVJ EC00652
SMOVL C00653 +MOVJ EC00653
SMOVL C00654 +MOVJ EC00654
SMOVL C00655 +MOVJ EC00655
SMOVL C00656 +MOVJ EC00656
SMOVL C00657 +MOVJ EC00657
SMOVL C00658 +MOVJ EC00658
SMOVL C00659 +MOVJ EC00659
SMOVL C00660 +MOVJ EC00660
SMOVL C00661 +MOVJ EC00661
SMOVL C00662 +MOVJ EC00662
SMOVL C00663 +MOVJ EC00663
SMOVL C00664 +MOVJ EC00664
SMOVL C00665 +MOVJ EC00665
SMOVL C00666 +MOVJ EC00666
SMOVL C00667 +MOVJ EC00667
SMOVL C00668 +MOVJ EC00668
SMOVL C00669 +MOVJ EC00669
SMOVL C00670 +MOVJ EC00670
SMOVL C00671 +MOVJ EC00671
SMOVL C00672 +MOVJ EC00672
SMOVL C00673 +MOVJ EC00673
SMOVL C00674 +MOVJ EC00674
SMOVL C00675 +MOVJ EC00675
SMOVL C00676 +MOVJ EC00676
SMOVL C00677 +MOVJ EC00677
SMOVL C00678 +MOVJ EC00678
SMOVL C00679 +MOVJ EC00679
SMOVL C00680 +MOVJ EC00680
SMOVL C00681 +MOVJ EC00681
SMOVL C00682 +MOVJ EC00682
SMOVL C00683 +MOVJ EC00683
SMOVL C00684 +MOVJ EC00684
SMOVL C00685 +MOVJ EC00685
SMOVL C00686 +MOVJ EC00686
SMOVL C00687 +MOVJ EC00687
SMOVL C00688 +MOVJ EC00688
SMOVL C00689 +MOVJ EC00689
SMOVL C00690 +MOVJ EC00690
SMOVL C00691 +MOVJ EC00691
SMOVL C00692 +MOVJ EC00692
SMOVL C00693 +MOVJ EC00693
SMOVL C00694 +MOVJ EC00694
SMOVL C00695 +MOVJ EC00695
SMOVL C00696 +MOVJ EC00696
SMOVL C00697 +MOVJ EC00697
SMOVL C00698 +MOVJ EC00698
SMOVL C00699 +MOVJ EC00699
SMOVL C00700 +MOVJ EC00700
SMOVL C00701 +MOVJ EC00701
SMOVL C00702 +MOVJ EC00702
SMOVL C00703 +MOVJ EC00703
SMOVL C00704 +MOVJ EC00704
SMOVL C00705 +MOVJ EC00705
SMOVL C00706 +MOVJ EC00706
SMOVL C00707 +MOVJ EC00707
SMOVL C00708 +MOVJ EC00708
SMOVL C00709 +MOVJ EC00709
SMOVL C00710 +MOVJ EC00710
SMOVL C00711 +MOVJ EC00711
SMOVL C00712 +MOVJ EC00712
SMOVL C00713 +MOVJ EC00713
SMOVL C00714 +MOVJ EC00714
SMOVL C00715 +MOVJ EC00715
SMOVL C00716 +MOVJ EC00716
SMOVL C00717 +MOVJ EC00717
SMOVL C00718 +MOVJ EC00718
SMOVL C00719 +MOVJ EC00719
SMOVL C00720 +MOVJ EC00720
SMOVL C00721 +MOVJ EC00721
SMOVL C00722 +MOVJ EC00722
SMOVL C00723 +MOVJ EC00723
SMOVL C00724 +MOVJ EC00724
SMOVL C00725 +MOVJ EC00725
SMOVL C00726 +MOVJ EC00726
SMOVL C00727 +MOVJ EC00727
SMOVL C00728 +MOVJ EC00728
SMOVL C00729 +MOVJ EC00729
SMOVL C00730 +MOVJ EC00730
SMOVL C00731 +MOVJ EC00731
SMOVL C00732 +MOVJ EC00732
SMOVL C00733 +MOVJ EC00733
SMOVL C00734 +MOVJ EC00734
SMOVL C00735 +MOVJ EC00735
SMOVL C00736 +MOVJ EC00736
SMOVL C00737 +MOVJ EC00737
SMOVL C00738 +MOVJ EC00738
SMOVL C00739 +MOVJ EC00739
SMOVL C00740 +MOVJ EC00740
SMOVL C00741 +MOVJ EC00741
SMOVL C00742 +MOVJ EC00742
SMOVL C00743 +MOVJ EC00743
SMOVL C00744 +MOVJ EC00744
SMOVL C00745 +MOVJ EC00745
SMOVL C00746 +MOVJ EC00746
SMOVL C00747 +MOVJ EC00747
SMOVL C00748 +MOVJ EC00748
SMOVL C00749 +MOVJ EC00749
SMOVL C00750 +MOVJ EC00750
SMOVL C00751 +MOVJ EC00751
SMOVL C00752 +MOVJ EC00752
SMOVL C00753 +MOVJ EC00753
SMOVL C00754 +MOVJ EC00754
SMOVL C00755 +MOVJ EC00755
SMOVL C00756 +MOVJ EC00756
SMOVL C00757 +MOVJ EC00757
SMOVL C00758 +MOVJ EC00758
SMOVL C00759 +MOVJ EC00759
SMOVL C00760 +MOVJ EC00760
SMOVL C00761 +MOVJ EC00761
SMOVL C00762 +MOVJ EC00762
SMOVL C00763 +MOVJ EC00763
SMOVL C00764 +MOVJ EC00764
SMOVL C00765 +MOVJ EC00765
SMOVL C00766 +MOVJ EC00766
SMOVL C00767 +MOVJ EC00767
SMOVL C00768 +MOVJ EC00768
SMOVL C00769 +MOVJ EC00769
SMOVL C00770 +MOVJ EC00770
SMOVL C00771 +MOVJ EC00771
SMOVL C00772 +MOVJ EC00772
SMOVL C00773 +MOVJ EC00773
SMOVL C00774 +MOVJ EC00774
SMOVL C00775 +MOVJ EC00775
SMOVL C00776 +MOVJ EC00776
SMOVL C00777 +MOVJ EC00777
SMOVL C00778 +MOVJ EC00778
SMOVL C00779 +MOVJ EC00779
SMOVL C00780 +MOVJ EC00780
SMOVL C00781 +MOVJ EC00781
SMOVL C00782 +MOVJ EC00782
SMOVL C00783 +MOVJ EC00783
SMOVL C00784 +MOVJ EC00784
SMOVL C00785 +MOVJ EC00785
SMOVL C00786 +MOVJ EC00786
SMOVL C00787 +MOVJ EC00787
SMOVL C00788 +MOVJ EC00788
SMOVL C00789 +MOVJ EC00789
SMOVL C00790 +MOVJ EC00790
SMOVL C00791 +MOVJ EC00791
SMOVL C00792 +MOVJ EC00792
SMOVL C00793 +MOVJ EC00793
SMOVL C00794 +MOVJ EC00794
SMOVL C00795 +MOVJ EC00795
SMOVL C00796 +MOVJ EC00796
SMOVL C00797 +MOVJ EC00797
SMOVL C00798 +MOVJ EC00798
SMOVL C00799 +MOVJ EC00799
SMOVL C00800 +MOVJ EC00800
SMOVL C00801 +MOVJ EC00801
SMOVL C00802 +MOVJ EC00802
SMOVL C00803 +MOVJ EC00803
SMOVL C00804 +MOVJ EC00804
SMOVL C00805 +MOVJ EC00805
SMOVL C00806 +MOVJ EC00806
SMOVL C00807 +MOVJ EC00807
SMOVL C00808 +MOVJ EC00808
SMOVL C00809 +MOVJ EC00809
SMOVL C00810 +MOVJ EC00810
SMOVL C00811 +MOVJ EC00811
SMOVL C00812 +MOVJ EC00812
SMOVL C00813 +MOVJ EC00813
SMOVL C00814 +MOVJ EC00814
SMOVL C00815 +MOVJ EC00815
SMOVL C00816 +MOVJ EC00816
SMOVL C00817 +MOVJ EC00817
SMOVL C00818 +MOVJ EC00818
SMOVL C00819 +MOVJ EC00819
SMOVL C00820 +MOVJ EC00820
SMOVL C00821 +MOVJ EC00821
SMOVL C00822 +MOVJ EC00822
SMOVL C00823 +MOVJ EC00823
SMOVL C00824 +MOVJ EC00824
SMOVL C00825 +MOVJ EC00825
SMOVL C00826 +MOVJ EC00826
SMOVL C00827 +MOVJ EC00827
SMOVL C00828 +MOVJ EC00828
SMOVL C00829 +MOVJ EC00829
SMOVL C00830 +MOVJ EC00830
SMOVL C00831 +MOVJ EC00831
SMOVL C00832 +MOVJ EC00832
SMOVL C00833 +MOVJ EC00833
SMOVL C00834 +MOVJ EC00834
SMOVL C00835 +MOVJ EC00835
SMOVL C00836 +MOVJ EC00836
SMOVL C00837 +MOVJ EC00837
SMOVL C00838 +MOVJ EC00838
SMOVL C00839 +MOVJ EC00839
SMOVL C00840 +MOVJ EC00840
SMOVL C00841 +MOVJ EC00841
SMOVL C00842 +MOVJ EC00842
SMOVL C00843 +MOVJ EC00843
SMOVL C00844 +MOVJ EC00844
SMOVL C00845 +MOVJ EC00845
SMOVL C00846 +MOVJ EC00846
SMOVL C00847 +MOVJ EC00847
SMOVL C00848 +MOVJ EC00848
SMOVL C00849 +MOVJ EC00849
SMOVL C00850 +MOVJ EC00850
SMOVL C00851 +MOVJ EC00851
SMOVL C00852 +MOVJ EC00852
SMOVL C00853 +MOVJ EC00853
SMOVL C00854 +MOVJ EC00854
SMOVL C00855 +MOVJ EC00855
SMOVL C00856 +MOVJ EC00856
SMOVL C00857 +MOVJ EC00857
SMOVL C00858 +MOVJ EC00858
SMOVL C00859 +MOVJ EC00859
SMOVL C00860 +MOVJ EC00860
SMOVL C00861 +MOVJ EC00861
SMOVL C00862 +MOVJ EC00862
SMOVL C00863 +MOVJ EC00863
SMOVL C00864 +MOVJ EC00864
SMOVL C00865 +MOVJ EC00865
SMOVL C00866 +MOVJ EC00866
SMOVL C00867 +MOVJ EC00867
SMOVL C00868 +MOVJ EC00868
SMOVL C00869 +MOVJ EC00869
SMOVL C00870 +MOVJ EC00870
SMOVL C00871 +MOVJ EC00871
SMOVL C00872 +MOVJ EC00872
SMOVL C00873 +MOVJ EC00873
SMOVL C00874 +MOVJ EC00874
SMOVL C00875 +MOVJ EC00875
SMOVL C00876 +MOVJ EC00876
SMOVL C00877 +MOVJ EC00877
SMOVL C00878 +MOVJ EC00878
SMOVL C00879 +MOVJ EC00879
SMOVL C00880 +MOVJ EC00880
SMOVL C00881 +MOVJ EC00881
SMOVL C00882 +MOVJ EC00882
SMOVL C00883 +MOVJ EC00883
SMOVL C00884 +MOVJ EC00884
SMOVL C00885 +MOVJ EC00885
SMOVL C00886 +MOVJ EC00886
SMOVL C00887 +MOVJ EC00887
SMOVL C00888 +MOVJ EC00888
SMOVL C00889 +MOVJ EC00889
SMOVL C00890 +MOVJ EC00890
SMOVL C00891 +MOVJ EC00891
SMOVL C00892 +MOVJ EC00892
SMOVL C00893 +MOVJ EC00893
SMOVL C00894 +MOVJ EC00894
SMOVL C00895 +MOVJ EC00895
SMOVL C00896 +MOVJ EC00896
SMOVL C00897 +MOVJ EC00897
SMOVL C00898 +MOVJ EC00898
SMOVL C00899 +MOVJ EC00899
SMOVL C00900 +MOVJ EC00900
SMOVL C00901 +MOVJ EC00901
SMOVL C00902 +MOVJ EC00902
SMOVL C00903 +MOVJ EC00903
SMOVL C00904 +MOVJ EC00904
SMOVL C00905 +MOVJ EC00905
SMOVL C00906 +MOVJ EC00906
SMOVL C00907 +MOVJ EC00907
SMOVL C00908 +MOVJ EC00908
SMOVL C00909 +MOVJ EC00909
SMOVL C00910 +MOVJ EC00910
SMOVL C00911 +MOVJ EC00911
SMOVL C00912 +MOVJ EC00912
SMOVL C00913 +MOVJ EC00913
SMOVL C00914 +MOVJ EC00914
SMOVL C00915 +MOVJ EC00915
SMOVL C00916 +MOVJ EC00916
SMOVL C00917 +MOVJ EC00917
SMOVL C00918 +MOVJ EC00918
SMOVL C00919 +MOVJ EC00919
SMOVL C00920 +MOVJ EC00920
SMOVL C00921 +MOVJ EC00921
SMOVL C00922 +MOVJ EC00922
SMOVL C00923 +MOVJ EC00923
SMOVL C00924 +MOVJ EC00924
SMOVL C00925 +MOVJ EC00925
SMOVL C00926 +MOVJ EC00926
SMOVL C00927 +MOVJ EC00927
SMOVL C00928 +MOVJ EC00928
SMOVL C00929 +MOVJ EC00929
SMOVL C00930 +MOVJ EC00930
SMOVL C00931 +MOVJ EC00931
SMOVL C00932 +MOVJ EC00932
SMOVL C00933 +MOVJ EC00933
SMOVL C00934 +MOVJ EC00934
SMOVL C00935 +MOVJ EC00935
SMOVL C00936 +MOVJ EC00936
SMOVL C00937 +MOVJ EC00937
SMOVL C00938 +MOVJ EC00938
SMOVL C00939 +MOVJ EC00939
SMOVL C00940 +MOVJ EC00940
SMOVL C00941 +MOVJ EC00941
SMOVL C00942 +MOVJ EC00942
SMOVL C00943 +MOVJ EC00943
SMOVL C00944 +MOVJ EC00944
SMOVL C00945 +MOVJ EC00945
SMOVL C00946 +MOVJ EC00946
SMOVL C00947 +MOVJ EC00947
SMOVL C00948 +MOVJ EC00948
SMOVL C00949 +MOVJ EC00949
SMOVL C00950 +MOVJ EC00950
SMOVL C00951 +MOVJ EC00951
SMOVL C00952 +MOVJ EC00952
SMOVL C00953 +MOVJ EC00953
SMOVL C00954 +MOVJ EC00954
SMOVL C00955 +MOVJ EC00955
SMOVL C00956 +MOVJ EC00956
SMOVL C00957 +MOVJ EC00957
SMOVL C00958 +MOVJ EC00958
SMOVL C00959 +MOVJ EC00959
SMOVL C00960 +MOVJ EC00960
SMOVL C00961 +MOVJ EC00961
SMOVL C00962 +MOVJ EC00962
SMOVL C00963 +MOVJ EC00963
SMOVL C00964 +MOVJ EC00964
SMOVL C00965 +MOVJ EC00965
SMOVL C00966 +MOVJ EC00966
SMOVL C00967 +MOVJ EC00967
SMOVL C00968 +MOVJ EC00968
SMOVL C00969 +MOVJ EC00969
SMOVL C00970 +MOVJ EC00970
SMOVL C00971 +MOVJ EC00971
SMOVL C00972 +MOVJ EC00972
SMOVL C00973 +MOVJ EC00973
SMOVL C00974 +MOVJ EC00974
SMOVL C00975 +MOVJ EC00975
SMOVL C00976 +MOVJ EC00976
SMOVL C00977 +MOVJ EC00977
SMOVL C00978 +MOVJ EC00978
SMOVL C00979 +MOVJ EC00979
SMOVL C00980 +MOVJ EC00980
SMOVL C00981 +MOVJ EC00981
SMOVL C00982 +MOVJ EC00982
SMOVL C00983 +MOVJ EC00983
SMOVL C00984 +MOVJ EC00984
SMOVL C00985 +MOVJ EC00985
SMOVL C00986 +MOVJ EC00986
SMOVL C00987 +MOVJ EC00987
SMOVL C00988 +MOVJ EC00988
SMOVL C00989 +MOVJ EC00989
SMOVL C00990 +MOVJ EC00990
SMOVL C00991 +MOVJ EC00991
SMOVL C00992 +MOVJ EC00992
SMOVL C00993 +MOVJ EC00993
SMOVL C00994 +MOVJ EC00994
SMOVL C00995 +MOVJ EC00995
SMOVL C00996 +MOVJ EC00996
SMOVL C00997 +MOVJ EC00997
SMOVL C00998 +MOVJ EC00998
SMOVL C00999 +MOVJ EC00999
SMOVL C01000 +MOVJ EC01000
SMOVL C01001 +MOVJ EC01001
SMOVL C01002 +MOVJ EC01002
SMOVL C01003 +MOVJ EC01003
SMOVL C01004 +MOVJ EC01004
SMOVL C01005 +MOVJ EC01005
SMOVL C01006 +MOVJ EC01006
SMOVL C01007 +MOVJ EC01007
SMOVL C01008 +MOVJ EC01008
SMOVL C01009 +MOVJ EC01009
SMOVL C01010 +MOVJ EC01010
SMOVL C01011 +MOVJ EC01011
SMOVL C01012 +MOVJ EC01012
SMOVL C01013 +MOVJ EC01013
SMOVL C01014 +MOVJ EC01014
SMOVL C01015 +MOVJ EC01015
SMOVL C01016 +MOVJ EC01016
SMOVL C01017 +MOVJ EC01017
SMOVL C01018 +MOVJ EC01018
SMOVL C01019 +MOVJ EC01019
SMOVL C01020 +MOVJ EC01020
SMOVL C01021 +MOVJ EC01021
SMOVL C01022 +MOVJ EC01022
SMOVL C01023 +MOVJ EC01023
SMOVL C01024 +MOVJ EC01024
SMOVL C01025 +MOVJ EC01025
SMOVL C01026 +MOVJ EC01026
SMOVL C01027 +MOVJ EC01027
SMOVL C01028 +MOVJ EC01028
SMOVL C01029 +MOVJ EC01029
SMOVL C01030 +MOVJ EC01030
SMOVL C01031 +MOVJ EC01031
SMOVL C01032 +MOVJ EC01032
SMOVL C01033 +MOVJ EC01033
SMOVL C01034 +MOVJ EC01034
SMOVL C01035 +MOVJ EC01035
SMOVL C01036 +MOVJ EC01036
SMOVL C01037 +MOVJ EC01037
SMOVL C01038 +MOVJ EC01038
SMOVL C01039 +MOVJ EC01039
SMOVL C01040 +MOVJ EC01040
SMOVL C01041 +MOVJ EC01041
SMOVL C01042 +MOVJ EC01042
SMOVL C01043 +MOVJ EC01043
SMOVL C01044 +MOVJ EC01044
SMOVL C01045 +MOVJ EC01045
SMOVL C01046 +MOVJ EC01046
SMOVL C01047 +MOVJ EC01047
SMOVL C01048 +MOVJ EC01048
SMOVL C01049 +MOVJ EC01049
SMOVL C01050 +MOVJ EC01050
SMOVL C01051 +MOVJ EC01051
SMOVL C01052 +MOVJ EC01052
SMOVL C01053 +MOVJ EC01053
SMOVL C01054 +MOVJ EC01054
SMOVL C01055 +MOVJ EC01055
SMOVL C01056 +MOVJ EC01056
SMOVL C01057 +MOVJ EC01057
SMOVL C01058 +MOVJ EC01058
SMOVL C01059 +MOVJ EC01059
SMOVL C01060 +MOVJ EC01060
SMOVL C01061 +MOVJ EC01061
SMOVL C01062 +MOVJ EC01062
SMOVL C01063 +MOVJ EC01063
SMOVL C01064 +MOVJ EC01064
SMOVL C01065 +MOVJ EC01065
SMOVL C01066 +MOVJ EC01066
SMOVL C01067 +MOVJ EC01067
SMOVL C01068 +MOVJ EC01068
SMOVL C01069 +MOVJ EC01069
SMOVL C01070 +MOVJ EC01070
SMOVL C01071 +MOVJ EC01071
SMOVL C01072 +MOVJ EC01072
SMOVL C01073 +MOVJ EC01073
SMOVL C01074 +MOVJ EC01074
SMOVL C01075 +MOVJ EC01075
SMOVL C01076 +MOVJ EC01076
SMOVL C01077 +MOVJ EC01077
SMOVL C01078 +MOVJ EC01078
SMOVL C01079 +MOVJ EC01079
SMOVL C01080 +MOVJ EC01080
SMOVL C01081 +MOVJ EC01081
SMOVL C01082 +MOVJ EC01082
SMOVL C01083 +MOVJ EC01083
SMOVL C01084 +MOVJ EC01084
SMOVL C01085 +MOVJ EC01085
SMOVL C01086 +MOVJ EC01086
SMOVL C01087 +MOVJ EC01087
SMOVL C01088 +MOVJ EC01088
SMOVL C01089 +MOVJ EC01089
SMOVL C01090 +MOVJ EC01090
SMOVL C01091 +MOVJ EC01091
SMOVL C01092 +MOVJ EC01092
SMOVL C01093 +MOVJ EC01093
SMOVL C01094 +MOVJ EC01094
SMOVL C01095 +MOVJ EC01095
SMOVL C01096 +MOVJ EC01096
SMOVL C01097 +MOVJ EC01097
SMOVL C01098 +MOVJ EC01098
SMOVL C01099 +MOVJ EC01099
SMOVL C01100 +MOVJ EC01100
SMOVL C01101 +MOVJ EC01101
SMOVL C01102 +MOVJ EC01102
SMOVL C01103 +MOVJ EC01103
SMOVL C01104 +MOVJ EC01104
SMOVL C01105 +MOVJ EC01105
SMOVL C01106 +MOVJ EC01106
SMOVL C01107 +MOVJ EC01107
SMOVL C01108 +MOVJ EC01108
SMOVL C01109 +MOVJ EC01109
SMOVL C01110 +MOVJ EC01110
SMOVL C01111 +MOVJ EC01111
SMOVL C01112 +MOVJ EC01112
SMOVL C01113 +MOVJ EC01113
SMOVL C01114 +MOVJ EC01114
SMOVL C01115 +MOVJ EC01115
SMOVL C01116 +MOVJ EC01116
SMOVL C01117 +MOVJ EC01117
SMOVL C01118 +MOVJ EC01118
SMOVL C01119 +MOVJ EC01119
SMOVL C01120 +MOVJ EC01120
SMOVL C01121 +MOVJ EC01121
SMOVL C01122 +MOVJ EC01122
SMOVL C01123 +MOVJ EC01123
SMOVL C01124 +MOVJ EC01124
SMOVL C01125 +MOVJ EC01125
SMOVL C01126 +MOVJ EC01126
SMOVL C01127 +MOVJ EC01127
SMOVL C01128 +MOVJ EC01128
SMOVL C01129 +MOVJ EC01129
SMOVL C01130 +MOVJ EC01130
SMOVL C01131 +MOVJ EC01131
SMOVL C01132 +MOVJ EC01132
SMOVL C01133 +MOVJ EC01133
SMOVL C01134 +MOVJ EC01134
SMOVL C01135 +MOVJ EC01135
SMOVL C01136 +MOVJ EC01136
SMOVL C01137 +MOVJ EC01137
SMOVL C01138 +MOVJ EC01138
SMOVL C01139 +MOVJ EC01139
SMOVL C01140 +MOVJ EC01140
SMOVL C01141 +MOVJ EC01141
SMOVL C01142 +MOVJ EC01142
SMOVL C01143 +MOVJ EC01143
SMOVL C01144 +MOVJ EC01144
SMOVL C01145 +MOVJ EC01145
SMOVL C01146 +MOVJ EC01146
SMOVL C01147 +MOVJ EC01147
SMOVL C01148 +MOVJ EC01148
SMOVL C01149 +MOVJ EC01149
SMOVL C01150 +MOVJ EC01150
SMOVL C01151 +MOVJ EC01151
SMOVL C01152 +MOVJ EC01152
SMOVL C01153 +MOVJ EC01153
SMOVL C01154 +MOVJ EC01154
SMOVL C01155 +MOVJ EC01155
SMOVL C01156 +MOVJ EC01156
SMOVL C01157 +MOVJ EC01157
SMOVL C01158 +MOVJ EC01158
SMOVL C01159 +MOVJ EC01159
SMOVL C01160 +MOVJ EC01160
SMOVL C01161 +MOVJ EC01161
SMOVL C01162 +MOVJ EC01162
SMOVL C01163 +MOVJ EC01163
SMOVL C01164 +MOVJ EC01164
SMOVL C01165 +MOVJ EC01165
SMOVL C01166 +MOVJ EC01166
SMOVL C01167 +MOVJ EC01167
SMOVL C01168 +MOVJ EC01168
SMOVL C01169 +MOVJ EC01169
SMOVL C01170 +MOVJ EC01170
SMOVL C01171 +MOVJ EC01171
SMOVL C01172 +MOVJ EC01172
SMOVL C01173 +MOVJ EC01173
SMOVL C01174 +MOVJ EC01174
SMOVL C01175 +MOVJ EC01175
SMOVL C01176 +MOVJ EC01176
SMOVL C01177 +MOVJ EC01177
SMOVL C01178 +MOVJ EC01178
SMOVL C01179 +MOVJ EC01179
SMOVL C01180 +MOVJ EC01180
SMOVL C01181 +MOVJ EC01181
SMOVL C01182 +MOVJ EC01182
SMOVL C01183 +MOVJ EC01183
SMOVL C01184 +MOVJ EC01184
SMOVL C01185 +MOVJ EC01185
SMOVL C01186 +MOVJ EC01186
SMOVL C01187 +MOVJ EC01187
SMOVL C01188 +MOVJ EC01188
SMOVL C01189 +MOVJ EC01189
SMOVL C01190 +MOVJ EC01190
SMOVL C01191 +MOVJ EC01191
SMOVL C01192 +MOVJ EC01192
SMOVL C01193 +MOVJ EC01193
SMOVL C01194 +MOVJ EC01194
SMOVL C01195 +MOVJ EC01195
SMOVL C01196 +MOVJ EC01196
SMOVL C01197 +MOVJ EC01197
SMOVL C01198 +MOVJ EC01198
SMOVL C01199 +MOVJ EC01199
SMOVL C01200 +MOVJ EC01200
SMOVL C01201 +MOVJ EC01201
SMOVL C01202 +MOVJ EC01202
SMOVL C01203 +MOVJ EC01203
SMOVL C01204 +MOVJ EC01204
SMOVL C01205 +MOVJ EC01205
SMOVL C01206 +MOVJ EC01206
SMOVL C01207 +MOVJ EC01207
SMOVL C01208 +MOVJ EC01208
SMOVL C01209 +MOVJ EC01209
SMOVL C01210 +MOVJ EC01210
SMOVL C01211 +MOVJ EC01211
SMOVL C01212 +MOVJ EC01212
SMOVL C01213 +MOVJ EC01213
SMOVL C01214 +MOVJ EC01214
SMOVL C01215 +MOVJ EC01215
SMOVL C01216 +MOVJ EC01216
SMOVL C01217 +MOVJ EC01217
SMOVL C01218 +MOVJ EC01218
SMOVL C01219 +MOVJ EC01219
SMOVL C01220 +MOVJ EC01220
SMOVL C01221 +MOVJ EC01221
SMOVL C01222 +MOVJ EC01222
SMOVL C01223 +MOVJ EC01223
SMOVL C01224 +MOVJ EC01224
SMOVL C01225 +MOVJ EC01225
SMOVL C01226 +MOVJ EC01226
SMOVL C01227 +MOVJ EC01227
SMOVL C01228 +MOVJ EC01228
SMOVL C01229 +MOVJ EC01229
SMOVL C01230 +MOVJ EC01230
SMOVL C01231 +MOVJ EC01231
SMOVL C01232 +MOVJ EC01232
SMOVL C01233 +MOVJ EC01233
SMOVL C01234 +MOVJ EC01234
SMOVL C01235 +MOVJ EC01235
SMOVL C01236 +MOVJ EC01236
SMOVL C01237 +MOVJ EC01237
SMOVL C01238 +MOVJ EC01238
SMOVL C01239 +MOVJ EC01239
SMOVL C01240 +MOVJ EC01240
SMOVL C01241 +MOVJ EC01241
SMOVL C01242 +MOVJ EC01242
SMOVL C01243 +MOVJ EC01243
SMOVL C01244 +MOVJ EC01244
SMOVL C01245 +MOVJ EC01245
SMOVL C01246 +MOVJ EC01246
SMOVL C01247 +MOVJ EC01247
SMOVL C01248 +MOVJ EC01248
SMOVL C01249 +MOVJ EC01249
SMOVL C01250 +MOVJ EC01250
SMOVL C01251 +MOVJ EC01251
SMOVL C01252 +MOVJ EC01252
SMOVL C01253 +MOVJ EC01253
SMOVL C01254 +MOVJ EC01254
SMOVL C01255 +MOVJ EC01255
SMOVL C01256 +MOVJ EC01256
SMOVL C01257 +MOVJ EC01257
SMOVL C01258 +MOVJ EC01258
SMOVL C01259 +MOVJ EC01259
SMOVL C01260 +MOVJ EC01260
SMOVL C01261 +MOVJ EC01261
SMOVL C01262 +MOVJ EC01262
SMOVL C01263 +MOVJ EC01263
SMOVL C01264 +MOVJ EC01264
SMOVL C01265 +MOVJ EC01265
SMOVL C01266 +MOVJ EC01266
SMOVL C01267 +MOVJ EC01267
SMOVL C01268 +MOVJ EC01268
SMOVL C01269 +MOVJ EC01269
SMOVL C01270 +MOVJ EC01270
SMOVL C01271 +MOVJ EC01271
SMOVL C01272 +MOVJ EC01272
SMOVL C01273 +MOVJ EC01273
SMOVL C01274 +MOVJ EC01274
SMOVL C01275 +MOVJ EC01275
SMOVL C01276 +MOVJ EC01276
SMOVL C01277 +MOVJ EC01277
SMOVL C01278 +MOVJ EC01278
SMOVL C01279 +MOVJ EC01279
SMOVL C01280 +MOVJ EC01280
SMOVL C01281 +MOVJ EC01281
SMOVL C01282 +MOVJ EC01282
SMOVL C01283 +MOVJ EC01283
SMOVL C01284 +MOVJ EC01284
SMOVL C01285 +MOVJ EC01285
SMOVL C01286 +MOVJ EC01286
SMOVL C01287 +MOVJ EC01287
SMOVL C01288 +MOVJ EC01288
SMOVL C01289 +MOVJ EC01289
SMOVL C01290 +MOVJ EC01290
SMOVL C01291 +MOVJ EC01291
SMOVL C01292 +MOVJ EC01292
SMOVL C01293 +MOVJ EC01293
SMOVL C01294 +MOVJ EC01294
SMOVL C01295 +MOVJ EC01295
SMOVL C01296 +MOVJ EC01296
SMOVL C01297 +MOVJ EC01297
SMOVL C01298 +MOVJ EC01298
SMOVL C01299 +MOVJ EC01299
SMOVL C01300 +MOVJ EC01300
SMOVL C01301 +MOVJ EC01301
SMOVL C01302 +MOVJ EC01302
SMOVL C01303 +MOVJ EC01303
SMOVL C01304 +MOVJ EC01304
SMOVL C01305 +MOVJ EC01305
SMOVL C01306 +MOVJ EC01306
SMOVL C01307 +MOVJ EC01307
SMOVL C01308 +MOVJ EC01308
SMOVL C01309 +MOVJ EC01309
SMOVL C01310 +MOVJ EC01310
SMOVL C01311 +MOVJ EC01311
SMOVL C01312 +MOVJ EC01312
SMOVL C01313 +MOVJ EC01313
SMOVL C01314 +MOVJ EC01314
SMOVL C01315 +MOVJ EC01315
SMOVL C01316 +MOVJ EC01316
SMOVL C01317 +MOVJ EC01317
SMOVL C01318 +MOVJ EC01318
SMOVL C01319 +MOVJ EC01319
SMOVL C01320 +MOVJ EC01320
SMOVL C01321 +MOVJ EC01321
SMOVL C01322 +MOVJ EC01322
SMOVL C01323 +MOVJ EC01323
SMOVL C01324 +MOVJ EC01324
SMOVL C01325 +MOVJ EC01325
SMOVL C01326 +MOVJ EC01326
SMOVL C01327 +MOVJ EC01327
SMOVL C01328 +MOVJ EC01328
SMOVL C01329 +MOVJ EC01329
SMOVL C01330 +MOVJ EC01330
SMOVL C01331 +MOVJ EC01331
SMOVL C01332 +MOVJ EC01332
SMOVL C01333 +MOVJ EC01333
SMOVL C01334 +MOVJ EC01334
SMOVL C01335 +MOVJ EC01335
SMOVL C01336 +MOVJ EC01336
SMOVL C01337 +MOVJ EC01337
SMOVL C01338 +MOVJ EC01338
SMOVL C01339 +MOVJ EC01339
SMOVL C01340 +MOVJ EC01340
SMOVL C01341 +MOVJ EC01341
SMOVL C01342 +MOVJ EC01342
SMOVL C01343 +MOVJ EC01343
SMOVL C01344 +MOVJ EC01344
SMOVL C01345 +MOVJ EC01345
SMOVL C01346 +MOVJ EC01346
SMOVL C01347 +MOVJ EC01347
SMOVL C01348 +MOVJ EC01348
SMOVL C01349 +MOVJ EC01349
SMOVL C01350 +MOVJ EC01350
SMOVL C01351 +MOVJ EC01351
SMOVL C01352 +MOVJ EC01352
SMOVL C01353 +MOVJ EC01353
SMOVL C01354 +MOVJ EC01354
